(* IEC 61131-3 sources: Industry-PLC-LLM/data/PLCBEAD_repo/PLCBEAD_PLCEmbed-main/PLC-BEAD/Source/OpenPLCv2, 619 files *)

(* ---- YAHOO_WEATHER_DESC_GE.ST ---- *)
TYPE
  oscat_STRING1               : STRING;
  oscat_STRING2               : STRING;
  oscat_STRING3               : STRING;
  oscat_STRING4               : STRING;
  oscat_STRING5               : STRING;
  oscat_STRING8               : STRING;
  oscat_STRING10              : STRING;
  oscat_STRING12            : STRING;
  oscat_STRING15            : STRING;
  oscat_STRING20            : STRING;
  oscat_STRING27            : STRING;
  oscat_STRING30            : STRING;
  oscat_STRING32            : STRING;
  oscat_STRING40            : STRING;
  oscat_STRING48            : STRING;
  oscat_STRING50            : STRING;
  oscat_STRING60            : STRING;
  oscat_STRING64            : STRING;
  oscat_STRING80            : STRING;
  oscat_STRING120            : STRING;
  oscat_STRING140            : STRING;
  oscat_STRING160            : STRING;
  oscat_STRING180            : STRING;
  oscat_STRING190            : STRING;
  oscat_STRING250            : STRING;
END_TYPE

TYPE
  oscat_IP_FIFO128_DATA  : ARRAY [1..128] OF BYTE;
  oscat_Mailbox  : ARRAY [1..16] OF BYTE;

  oscat_IP_FIFO_DATA :
  STRUCT
	X       : oscat_IP_FIFO128_DATA; (* IP_ID FIFO Speicher          *)
	Y       : oscat_IP_FIFO128_DATA; (* IP_ID Z�hler                 *)
	ID      : BYTE;                  (* h�chste vergabene id         *)
	MAX_ID  : BYTE;                  (* maximal Anmeldungen pro ID   *)
    INIT    : BOOL;                  (* Initialisierung durchgef�hrt *)
	EMPTY   : BOOL;                  (* FIFO leer                    *)
	FULL    : BOOL;                  (* FIFO voll                    *)
	TOP     : INT;                   (* maximale anzahl in FIFO      *)
	NW      : INT;                   (* Schreibzeiger                *)
	NR      : INT;                   (* Lesezeiger                   *)
  END_STRUCT;

  oscat_IP_C:
  STRUCT
  	C_MODE:			BYTE;          		(*W Mode: TCP/UCP AKTIV/PASSIV                               *)
	C_PORT:         WORD;          		(*W Portnummer                                               *)
	C_IP:           DWORD;         		(*W IP-Adresse gepackt wwxxyyzz = www.xxx.yyy.zzz            *)
    C_STATE:        BYTE;          		(*R Verbindungsstatus ON/OFF + Flanke ON/OFF                 *)
	C_ENABLE:       BOOL;          		(*W Freigabe f�r Connect                                     *)
    R_OBSERVE:      BOOL;          		(*W Empfang ueberwachen                                      *)
    TIME_RESET:     BOOL;          		(*W Alle Timer ruecksetzen                                   *)
	ERROR:          DWORD;         		(*R vvwwxxyy (vv = CON_ERROR, ww = SEN_ERROR, xx = REC_ERROR *)
    FIFO:           oscat_IP_FIFO_DATA; (*I IP FIFO Struktur                                         *)
	MAILBOX:		oscat_Mailbox;		(*I Mailbox: Datenbereich f�r Bausteindatenaustausch         *)
  END_STRUCT;

  oscat_XML_CONTROL:
  STRUCT
    COMMAND:             WORD;            (*W                 *)
    WATCHDOG:            TIME;            (*W                 *)
    START_POS:           UINT;            (*W                 *)
    STOP_POS:            UINT;            (*W                 *)
    COUNT:               UINT;            (*R                 *)
    TYP:                 INT;             (*R                 *)
    LEVEL:               UINT;            (*R                 *)
    PATH:                oscat_STRING250; (*R                 *)
    ELEMENT:             oscat_STRING250; (*R                 *)
    ATTRIBUTE:           oscat_STRING250; (*R                 *)
    VALUE:               oscat_STRING250; (*R                 *)
    BLOCK1_START:        UINT;            (*R                 *)
    BLOCK1_STOP:         UINT;            (*R                 *)
    BLOCK2_START:        UINT;            (*R                 *)
    BLOCK2_STOP:         UINT;            (*R                 *)
  END_STRUCT;

  (* --------- WORLD WEATHER --------- *)

  oscat_WORLD_WEATHER_CUR :
  STRUCT
	OBSERVATION_TIME : oscat_STRING8;
	TEMP_C           : INT;
	WEATHER_CODE     : INT;
	WEATHER_DESC 	 : oscat_STRING60;
	WEATHER_ICON     : INT;
	WIND_SPEED_MILES : INT;
	WIND_SPEED_KMPH  : INT;
	WIND_DIR_DEGREE  : INT;
	WIND_DIR16POINT  : oscat_STRING3;
	PRECIPMM         : REAL;
	HUMIDITY         : INT;
	VISIBILITY       : INT;
	PRESSURE         : INT;
	CLOUDOVER        : INT;
  END_STRUCT;

  oscat_WORLD_WEATHER_DAY :
  STRUCT
	DATE_OF_DAY      : oscat_STRING10;
	TEMP_MAX_C       : INT;
	TEMP_MAX_F       : INT;
	TEMP_MIN_C       : INT;
	TEMP_MIN_F       : INT;
	WIND_SPEED_MILES : INT;
	WIND_SPEED_KMPH  : INT;
	WIND_DIR_DEGREE  : INT;
	WIND_DIR16POINT  : oscat_STRING3;
	WEATHER_CODE     : INT;
	WEATHER_DESC     : oscat_STRING60;
	WEATHER_ICON     : INT;
	PRECIPMM         : REAL;
  END_STRUCT;

  oscat_WORLD_WEATHER_DAY_ARR : ARRAY [0..4] OF oscat_WORLD_WEATHER_DAY;

  oscat_WORLD_WEATHER_DATA :
  STRUCT
	CUR : oscat_WORLD_WEATHER_CUR;
	DAY : oscat_WORLD_WEATHER_DAY_ARR;
  END_STRUCT;

  oscat_WORLD_WEATHER_aI0_41 : ARRAY[0..41] OF INT;

  (* --------- WEATHER CHANNEL --------- *)
  oscat_YAHOO_WEATHER_DATA:
  STRUCT
    TIMETOLIVE:                 INT;              (* TIME TO LIVE: HOW LONG IN MINUTES THIS FEED SHOULD BE CACHED         *)
    LOCATION_CITY:              OSCAT_STRING40;   (* THE LOCATION OF THIS FORECAST: CITY: CITY NAME  *)
    LOCATION_REGION:            OSCAT_STRING20;   (* THE LOCATION OF THIS FORECAST: REGION: STATE, TERRITORY, OR REGION, IF GIVEN *)
    LOCATION_COUNTRY:           OSCAT_STRING20;    (* THE LOCATION OF THIS FORECAST: COUNTRY: TWO-CHARACTER COUNTRY CODE *)
    UNIT_TEMPERATURE:           OSCAT_STRING1;    (* TEMPERATURE: DEGREE UNITS, F FOR FAHRENHEIT OR C FOR CELSIUS *)
    UNIT_DISTANCE:              OSCAT_STRING2;    (* DISTANCE: UNITS FOR DISTANCE, MI FOR MILES OR KM FOR KILOMETERS *)
    UNIT_PRESSURE:              OSCAT_STRING2;    (* PRESSURE: UNITS OF BAROMETRIC PRESSURE, IN FOR POUNDS PER SQUARE INCH OR MB FOR MILLIBARS *)
    UNIT_SPEED:                 OSCAT_STRING4;    (* SPEED: UNITS OF SPEED, MPH FOR MILES PER HOUR OR KPH FOR KILOMETERS PER HOUR *)
    WIND_CHILL:                 INT;              (* FORECAST INFORMATION ABOUT WIND CHILL IN DEGREES *)
    WIND_DIRECTION:             INT;              (* FORECAST INFORMATION ABOUT WIND DIRECTION, IN DEGREES *)
    WIND_SPEED:                 REAL;             (* FORECAST INFORMATION ABOUT WIND SPEED, IN THE UNITS (MPH OR KPH)*)
    ATMOSPHERE_HUMIDITY:        INT;              (* FORECAST INFORMATION ABOUT CURRENT ATMOSPHERIC HUMIDITY: HUMIDITY, IN PERCENT  *)
    ATMOSPHERE_PRESSURE:        INT;              (* FORECAST INFORMATION ABOUT CURRENT ATMOSPHERIC PRESSURE: BAROMETRIC PRESSURE, IN THE UNITS (IN OR MB) *)
	ATMOSPHERE_VISIBILITY:      REAL;             (* FORECAST INFORMATION ABOUT CURRENT ATMOSPHERIC VISIBILITY, IN THE UNITS (MI OR KM) *)
	ATMOSPHERE_RISING:          INT;              (* FORECAST INFORMATION ABOUT RISING: STATE OF THE BAROMETRIC PRESSURE: STEADY (0), RISING (1), OR FALLING (2). (INTEGER: 0, 1, 2) *)
    ASTRONOMY_SUNRISE:          OSCAT_STRING10;   (* SUNRISE: TODAY'S SUNRISE TIME. THE TIME IS A STRING IN A LOCAL TIME FORMAT OF "H:MM AM/PM" *)
    ASTRONOMY_SUNSET:           OSCAT_STRING10;   (* SUNSET: TODAY'S SUNSET TIME. THE TIME IS A STRING IN A LOCAL TIME FORMAT OF "H:MM AM/PM", *)
    GEO_LATITUDE:               REAL;             (* THE LATITUDE OF THE LOCATION *)
    GEO_LONGITUDE:              REAL;             (* THE LONGITUDE OF THE LOCATION *)
    CUR_CONDITIONS_TEMP:        INT;              (* THE CURRENT WEATHER CONDITIONS: TEMP: THE CURRENT TEMPERATURE, IN THE UNITS (F OR C) *)
    CUR_CONDITIONS_TEXT:        OSCAT_STRING40;   (* THE CURRENT WEATHER CONDITIONS: TEXT: A TEXTUAL DESCRIPTION OF CONDITIONS *)
    CUR_CONDITIONS_CODE:        INT;              (* THE CURRENT WEATHER CONDITIONS: CODE: THE CONDITION CODE FOR THIS FORECAST *)
	CUR_CONDITIONS_ICON:        INT;			  (* THE CURRENT WEATHER CONDITIONS: ICON: THE CONDITION ICON FOR THIS FORECAST *)
    FORCAST_TODAY_LOW_TEMP:     INT;              (* THE FORCAST TODAY WEATHER CONDITIONS: THE FORECASTED LOW TEMPERATURE FOR THIS DAY IN THE UNITS (F OR C) *)
    FORCAST_TODAY_HIGH_TEMP:    INT;              (* THE FORCAST TODAY WEATHER CONDITIONS: THE FORECASTED HIGH TEMPERATURE FOR THIS DAY IN THE UNITS (F OR C) *)
    FORCAST_TODAY_TEXT:         OSCAT_STRING40;   (* THE FORCAST TODAY WEATHER CONDITIONS: TEXT: A TEXTUAL DESCRIPTION OF CONDITIONS *)
    FORCAST_TODAY_CODE:         INT;              (* THE CURRENT WEATHER CONDITIONS: CODE: THE CONDITION CODE FOR THIS FORECAST *)
	FORCAST_TODAY_ICON:         INT;			  (* THE CURRENT WEATHER CONDITIONS: ICON: THE CONDITION ICON FOR THIS FORECAST *)
    FORCAST_TOMORROW_LOW_TEMP:  INT;              (* THE FORCAST TOMORROW WEATHER CONDITIONS: THE FORECASTED LOW TEMPERATURE FOR THIS DAY IN THE UNITS (F OR C) *)
    FORCAST_TOMORROW_HIGH_TEMP: INT;              (* THE FORCAST TOMORROW WEATHER CONDITIONS: THE FORECASTED HIGH TEMPERATURE FOR THIS DAY IN THE UNITS (F OR C) *)
    FORCAST_TOMORROW_TEXT:      OSCAT_STRING40;   (* THE FORCAST TOMORROW WEATHER CONDITIONS: TEXT: A TEXTUAL DESCRIPTION OF CONDITIONS *)
    FORCAST_TOMORROW_CODE:      INT;              (* THE CURRENT WEATHER CONDITIONS: CODE: THE CONDITION CODE FOR THIS FORECAST *)
	FORCAST_TOMORROW_ICON:      INT;			  (* THE CURRENT WEATHER CONDITIONS: ICON: THE CONDITION ICON FOR THIS FORECAST *)
  END_STRUCT;

  oscat_YAHOO_WEATHER_aI0_48 : ARRAY[0..48] OF INT;

  oscat_IP2GEO_DATA:
  STRUCT
	STATE :				BOOL;			  (* STATE *)
	IP4 :				DWORD;			  (* IP-Adresse *)
    COUNTRY_CODE :		oscat_STRING2;    (*   *)
    COUNTRY_NAME :		oscat_STRING20;   (*   *)
    REGION_CODE :		oscat_STRING2;    (*   *)
    REGION_NAME :		oscat_STRING20;   (*   *)
    CITY :				oscat_STRING20;   (*   *)
    GEO_LATITUDE :		REAL;             (*   *)
    GEO_LONGITUDE :		REAL;             (*   *)
	TIME_ZONE_NAME :	oscat_STRING20;
	GMT_OFFSET :		INT;
	IS_DST :			BOOL;
  END_STRUCT;
END_TYPE

FUNCTION_BLOCK YAHOO_WEATHER_DESC_GE_Block

	VAR_INPUT
		ACTIVATE :	BOOL;
	END_VAR

	VAR_IN_OUT
		YW :	oscat_YAHOO_WEATHER_DATA;
	END_VAR

	VAR
		act_last :	BOOL;
		x :	INT;
		y :	INT;
		str :	oscat_STRING40;
	END_VAR

	IF ACTIVATE AND act_last = FALSE THEN
		FOR y := 1 TO 4 DO
			CASE y OF
			1:	x := YW.CUR_CONDITIONS_CODE;
			2 :	YW.CUR_CONDITIONS_TEXT := str;
				x := YW.FORCAST_TODAY_CODE;
			3 :	YW.FORCAST_TODAY_TEXT := str;
				x := YW.FORCAST_TOMORROW_CODE;
			4 :	YW.FORCAST_TOMORROW_TEXT := str;
			END_CASE;

			CASE x OF
			00:	str := 'Wirbelsturm';
			01:	str := 'Tropensturm';
			02:	str := 'Wirbelsturm';
			03:	str := 'starkes Gewitter ';
			04:	str := 'Gewitter';
			05:	str := 'Schneeregen';
			06:	str := 'Schneeregen';
			07:	str := 'Schneeregen';
			08:	str := 'gefrierender Nieselregen';
			09:	str := 'Nieselregen';
			10:	str := 'gefrierender Regen';
			11:	str := 'sertsehn';
			12:	str := 'sertstrets';
			13:	str := 'sjstj';
			14:	str := 'leichte yrderew';
			15:	str := 'Schneetreiben';
			16:	str := 'Schnee';
			17:	str := 'Hagel';
			18:	str := 'Schneeregen';
			19:	str := 'Staub';
			20:	str := 'nebelig';
			21:	str := 'Dunst';
			22:	str := 'rauchig';
			23:	str := 'sertsert';
			24:	str := 'windig';
			25:	str := 'kalt';
			26:	str := 'sertsert';
			27:	str := 'meist sertsert';
			28:	str := 'meist sertsert';
			29:	str := 'teilweise serhser';
			30:	str := 'teilweise sertsertshe';
			31:	str := 'klar';
			32:	str := 'sonnig';
			33:	str := 'heiter';
			34:	str := 'heiter';
			35:	str := 'Regen und Hagel';
			36:	str := 'WRYTWRYH';
			37:	str := 'esrertsertr';
			38:	str := 'vereinzelte Gewitter';
			39:	str := 'vereinzelte Gewitter';
			40:	str := 'verteesr';
			41:	str := 'sjstjtj';
			42:	str := 'sertsert';
			43:	str := 'sertsert';
			44:	str := 'sertsert';
			45:	str := 'sertsert';
			46:	str := 'sertsert';
			47:	str := 'srtsert';
			ELSE
				str := 'sertsert';
			END_CASE;
		END_FOR;
	END_IF;
	act_last := ACTIVATE;

END_FUNCTION_BLOCK

PROGRAM program0
	VAR
		ACTIVATE :	BOOL;
		YW :	oscat_YAHOO_WEATHER_DATA;

		func_block : YAHOO_WEATHER_DESC_GE_Block;
	END_VAR
	func_block.ACTIVATE := ACTIVATE;
	func_block.YW := YW;

	func_block();
	YW  := func_block.YW;
END_PROGRAM

CONFIGURATION Config0
	RESOURCE Res0 ON PLC
		TASK task0(INTERVAL := T#20ms,PRIORITY := 0);
		PROGRAM instance0 WITH task0 : program0;
	END_RESOURCE
END_CONFIGURATION

(* ---- YAHOO_WEATHER_ICON_OSCAT.ST ---- *)
TYPE
  oscat_STRING1               : STRING;
  oscat_STRING2               : STRING;
  oscat_STRING3               : STRING;
  oscat_STRING4               : STRING;
  oscat_STRING5               : STRING;
  oscat_STRING8               : STRING;
  oscat_STRING10              : STRING;
  oscat_STRING12            : STRING;
  oscat_STRING15            : STRING;
  oscat_STRING20            : STRING;
  oscat_STRING27            : STRING;
  oscat_STRING30            : STRING;
  oscat_STRING32            : STRING;
  oscat_STRING40            : STRING;
  oscat_STRING48            : STRING;
  oscat_STRING50            : STRING;
  oscat_STRING60            : STRING;
  oscat_STRING64            : STRING;
  oscat_STRING80            : STRING;
  oscat_STRING120            : STRING;
  oscat_STRING140            : STRING;
  oscat_STRING160            : STRING;
  oscat_STRING180            : STRING;
  oscat_STRING190            : STRING;
  oscat_STRING250            : STRING;
END_TYPE

TYPE
  oscat_IP_FIFO128_DATA  : ARRAY [1..128] OF BYTE;
  oscat_Mailbox  : ARRAY [1..16] OF BYTE;

  oscat_IP_FIFO_DATA :
  STRUCT
	X       : oscat_IP_FIFO128_DATA; (* IP_ID FIFO Speicher          *)
	Y       : oscat_IP_FIFO128_DATA; (* IP_ID Z�hler                 *)
	ID      : BYTE;                  (* h�chste vergabene id         *)
	MAX_ID  : BYTE;                  (* maximal Anmeldungen pro ID   *)
    INIT    : BOOL;                  (* Initialisierung durchgef�hrt *)
	EMPTY   : BOOL;                  (* FIFO leer                    *)
	FULL    : BOOL;                  (* FIFO voll                    *)
	TOP     : INT;                   (* maximale anzahl in FIFO      *)
	NW      : INT;                   (* Schreibzeiger                *)
	NR      : INT;                   (* Lesezeiger                   *)
  END_STRUCT;

  oscat_IP_C:
  STRUCT
  	C_MODE:			BYTE;          		(*W Mode: TCP/UCP AKTIV/PASSIV                               *)
	C_PORT:         WORD;          		(*W Portnummer                                               *)
	C_IP:           DWORD;         		(*W IP-Adresse gepackt wwxxyyzz = www.xxx.yyy.zzz            *)
    C_STATE:        BYTE;          		(*R Verbindungsstatus ON/OFF + Flanke ON/OFF                 *)
	C_ENABLE:       BOOL;          		(*W Freigabe f�r Connect                                     *)
    R_OBSERVE:      BOOL;          		(*W Empfang ueberwachen                                      *)
    TIME_RESET:     BOOL;          		(*W Alle Timer ruecksetzen                                   *)
	ERROR:          DWORD;         		(*R vvwwxxyy (vv = CON_ERROR, ww = SEN_ERROR, xx = REC_ERROR *)
    FIFO:           oscat_IP_FIFO_DATA; (*I IP FIFO Struktur                                         *)
	MAILBOX:		oscat_Mailbox;		(*I Mailbox: Datenbereich f�r Bausteindatenaustausch         *)
  END_STRUCT;

  oscat_XML_CONTROL:
  STRUCT
    COMMAND:             WORD;            (*W                 *)
    WATCHDOG:            TIME;            (*W                 *)
    START_POS:           UINT;            (*W                 *)
    STOP_POS:            UINT;            (*W                 *)
    COUNT:               UINT;            (*R                 *)
    TYP:                 INT;             (*R                 *)
    LEVEL:               UINT;            (*R                 *)
    PATH:                oscat_STRING250; (*R                 *)
    ELEMENT:             oscat_STRING250; (*R                 *)
    ATTRIBUTE:           oscat_STRING250; (*R                 *)
    VALUE:               oscat_STRING250; (*R                 *)
    BLOCK1_START:        UINT;            (*R                 *)
    BLOCK1_STOP:         UINT;            (*R                 *)
    BLOCK2_START:        UINT;            (*R                 *)
    BLOCK2_STOP:         UINT;            (*R                 *)
  END_STRUCT;

  (* --------- WORLD WEATHER --------- *)

  oscat_WORLD_WEATHER_CUR :
  STRUCT
	OBSERVATION_TIME : oscat_STRING8;
	TEMP_C           : INT;
	WEATHER_CODE     : INT;
	WEATHER_DESC 	 : oscat_STRING60;
	WEATHER_ICON     : INT;
	WIND_SPEED_MILES : INT;
	WIND_SPEED_KMPH  : INT;
	WIND_DIR_DEGREE  : INT;
	WIND_DIR16POINT  : oscat_STRING3;
	PRECIPMM         : REAL;
	HUMIDITY         : INT;
	VISIBILITY       : INT;
	PRESSURE         : INT;
	CLOUDOVER        : INT;
  END_STRUCT;

  oscat_WORLD_WEATHER_DAY :
  STRUCT
	DATE_OF_DAY      : oscat_STRING10;
	TEMP_MAX_C       : INT;
	TEMP_MAX_F       : INT;
	TEMP_MIN_C       : INT;
	TEMP_MIN_F       : INT;
	WIND_SPEED_MILES : INT;
	WIND_SPEED_KMPH  : INT;
	WIND_DIR_DEGREE  : INT;
	WIND_DIR16POINT  : oscat_STRING3;
	WEATHER_CODE     : INT;
	WEATHER_DESC     : oscat_STRING60;
	WEATHER_ICON     : INT;
	PRECIPMM         : REAL;
  END_STRUCT;

  oscat_WORLD_WEATHER_DAY_ARR : ARRAY [0..4] OF oscat_WORLD_WEATHER_DAY;

  oscat_WORLD_WEATHER_DATA :
  STRUCT
	CUR : oscat_WORLD_WEATHER_CUR;
	DAY : oscat_WORLD_WEATHER_DAY_ARR;
  END_STRUCT;

  oscat_WORLD_WEATHER_aI0_41 : ARRAY[0..41] OF INT;

  (* --------- WEATHER CHANNEL --------- *)
  oscat_YAHOO_WEATHER_DATA:
  STRUCT
    TIMETOLIVE:                 INT;              (* TIME TO LIVE: HOW LONG IN MINUTES THIS FEED SHOULD BE CACHED         *)
    LOCATION_CITY:              OSCAT_STRING40;   (* THE LOCATION OF THIS FORECAST: CITY: CITY NAME  *)
    LOCATION_REGION:            OSCAT_STRING20;   (* THE LOCATION OF THIS FORECAST: REGION: STATE, TERRITORY, OR REGION, IF GIVEN *)
    LOCATION_COUNTRY:           OSCAT_STRING20;    (* THE LOCATION OF THIS FORECAST: COUNTRY: TWO-CHARACTER COUNTRY CODE *)
    UNIT_TEMPERATURE:           OSCAT_STRING1;    (* TEMPERATURE: DEGREE UNITS, F FOR FAHRENHEIT OR C FOR CELSIUS *)
    UNIT_DISTANCE:              OSCAT_STRING2;    (* DISTANCE: UNITS FOR DISTANCE, MI FOR MILES OR KM FOR KILOMETERS *)
    UNIT_PRESSURE:              OSCAT_STRING2;    (* PRESSURE: UNITS OF BAROMETRIC PRESSURE, IN FOR POUNDS PER SQUARE INCH OR MB FOR MILLIBARS *)
    UNIT_SPEED:                 OSCAT_STRING4;    (* SPEED: UNITS OF SPEED, MPH FOR MILES PER HOUR OR KPH FOR KILOMETERS PER HOUR *)
    WIND_CHILL:                 INT;              (* FORECAST INFORMATION ABOUT WIND CHILL IN DEGREES *)
    WIND_DIRECTION:             INT;              (* FORECAST INFORMATION ABOUT WIND DIRECTION, IN DEGREES *)
    WIND_SPEED:                 REAL;             (* FORECAST INFORMATION ABOUT WIND SPEED, IN THE UNITS (MPH OR KPH)*)
    ATMOSPHERE_HUMIDITY:        INT;              (* FORECAST INFORMATION ABOUT CURRENT ATMOSPHERIC HUMIDITY: HUMIDITY, IN PERCENT  *)
    ATMOSPHERE_PRESSURE:        INT;              (* FORECAST INFORMATION ABOUT CURRENT ATMOSPHERIC PRESSURE: BAROMETRIC PRESSURE, IN THE UNITS (IN OR MB) *)
	ATMOSPHERE_VISIBILITY:      REAL;             (* FORECAST INFORMATION ABOUT CURRENT ATMOSPHERIC VISIBILITY, IN THE UNITS (MI OR KM) *)
	ATMOSPHERE_RISING:          INT;              (* FORECAST INFORMATION ABOUT RISING: STATE OF THE BAROMETRIC PRESSURE: STEADY (0), RISING (1), OR FALLING (2). (INTEGER: 0, 1, 2) *)
    ASTRONOMY_SUNRISE:          OSCAT_STRING10;   (* SUNRISE: TODAY'S SUNRISE TIME. THE TIME IS A STRING IN A LOCAL TIME FORMAT OF "H:MM AM/PM" *)
    ASTRONOMY_SUNSET:           OSCAT_STRING10;   (* SUNSET: TODAY'S SUNSET TIME. THE TIME IS A STRING IN A LOCAL TIME FORMAT OF "H:MM AM/PM", *)
    GEO_LATITUDE:               REAL;             (* THE LATITUDE OF THE LOCATION *)
    GEO_LONGITUDE:              REAL;             (* THE LONGITUDE OF THE LOCATION *)
    CUR_CONDITIONS_TEMP:        INT;              (* THE CURRENT WEATHER CONDITIONS: TEMP: THE CURRENT TEMPERATURE, IN THE UNITS (F OR C) *)
    CUR_CONDITIONS_TEXT:        OSCAT_STRING40;   (* THE CURRENT WEATHER CONDITIONS: TEXT: A TEXTUAL DESCRIPTION OF CONDITIONS *)
    CUR_CONDITIONS_CODE:        INT;              (* THE CURRENT WEATHER CONDITIONS: CODE: THE CONDITION CODE FOR THIS FORECAST *)
	CUR_CONDITIONS_ICON:        INT;			  (* THE CURRENT WEATHER CONDITIONS: ICON: THE CONDITION ICON FOR THIS FORECAST *)
    FORCAST_TODAY_LOW_TEMP:     INT;              (* THE FORCAST TODAY WEATHER CONDITIONS: THE FORECASTED LOW TEMPERATURE FOR THIS DAY IN THE UNITS (F OR C) *)
    FORCAST_TODAY_HIGH_TEMP:    INT;              (* THE FORCAST TODAY WEATHER CONDITIONS: THE FORECASTED HIGH TEMPERATURE FOR THIS DAY IN THE UNITS (F OR C) *)
    FORCAST_TODAY_TEXT:         OSCAT_STRING40;   (* THE FORCAST TODAY WEATHER CONDITIONS: TEXT: A TEXTUAL DESCRIPTION OF CONDITIONS *)
    FORCAST_TODAY_CODE:         INT;              (* THE CURRENT WEATHER CONDITIONS: CODE: THE CONDITION CODE FOR THIS FORECAST *)
	FORCAST_TODAY_ICON:         INT;			  (* THE CURRENT WEATHER CONDITIONS: ICON: THE CONDITION ICON FOR THIS FORECAST *)
    FORCAST_TOMORROW_LOW_TEMP:  INT;              (* THE FORCAST TOMORROW WEATHER CONDITIONS: THE FORECASTED LOW TEMPERATURE FOR THIS DAY IN THE UNITS (F OR C) *)
    FORCAST_TOMORROW_HIGH_TEMP: INT;              (* THE FORCAST TOMORROW WEATHER CONDITIONS: THE FORECASTED HIGH TEMPERATURE FOR THIS DAY IN THE UNITS (F OR C) *)
    FORCAST_TOMORROW_TEXT:      OSCAT_STRING40;   (* THE FORCAST TOMORROW WEATHER CONDITIONS: TEXT: A TEXTUAL DESCRIPTION OF CONDITIONS *)
    FORCAST_TOMORROW_CODE:      INT;              (* THE CURRENT WEATHER CONDITIONS: CODE: THE CONDITION CODE FOR THIS FORECAST *)
	FORCAST_TOMORROW_ICON:      INT;			  (* THE CURRENT WEATHER CONDITIONS: ICON: THE CONDITION ICON FOR THIS FORECAST *)
  END_STRUCT;

  oscat_YAHOO_WEATHER_aI0_48 : ARRAY[0..48] OF INT;

  oscat_IP2GEO_DATA:
  STRUCT
	STATE :				BOOL;			  (* STATE *)
	IP4 :				DWORD;			  (* IP-Adresse *)
    COUNTRY_CODE :		oscat_STRING2;    (*   *)
    COUNTRY_NAME :		oscat_STRING20;   (*   *)
    REGION_CODE :		oscat_STRING2;    (*   *)
    REGION_NAME :		oscat_STRING20;   (*   *)
    CITY :				oscat_STRING20;   (*   *)
    GEO_LATITUDE :		REAL;             (*   *)
    GEO_LONGITUDE :		REAL;             (*   *)
	TIME_ZONE_NAME :	oscat_STRING20;
	GMT_OFFSET :		INT;
	IS_DST :			BOOL;
  END_STRUCT;
END_TYPE

FUNCTION_BLOCK YAHOO_WEATHER_ICON_OSCAT_Block

	VAR_INPUT
		ACTIVATE :	BOOL;
	END_VAR

	VAR_IN_OUT
		YW :	oscat_YAHOO_WEATHER_DATA;
	END_VAR

	VAR
		act_last :	BOOL;
		x :	INT;
		init :	BOOL;
		dat :	oscat_YAHOO_WEATHER_aI0_48;
	END_VAR

	IF not init THEN
		init := TRUE;

		dat[00] := 4;
		dat[01] := 2;
		dat[02] := 2;
		dat[03] := 4;
		dat[04] := 17;
		dat[05] := 1;
		dat[06] := 3;
		dat[07] := 1;
		dat[08] := 2;
		dat[09] := 2;
		dat[10] := 2;
		dat[11] := 2;
		dat[12] := 2;
		dat[13] := 3;
		dat[14] := 3;
		dat[15] := 3;
		dat[16] := 3;
		dat[17] := 5;
		dat[18] := 3;
		dat[19] := 6;
		dat[20] := 7;
		dat[21] := 14;
		dat[22] := 8;
		dat[23] := 9;
		dat[24] := 9;
		dat[25] := 10;
		dat[26] := 9;
		dat[27] := 11;
		dat[28] := 12;
		dat[29] := 11;
		dat[30] := 12;
		dat[31] := 13;
		dat[32] := 14;
		dat[33] := 15;
		dat[34] := 16;
		dat[35] := 4;
		dat[36] := 14;
		dat[37] := 4;
		dat[38] := 17;
		dat[39] := 2;
		dat[40] := 2;
		dat[41] := 3;
		dat[42] := 3;
		dat[43] := 3;
		dat[44] := 12;
		dat[45] := 2;
		dat[46] := 3;
		dat[47] := 4;
		dat[48] := 0;
	END_IF;

	IF ACTIVATE AND act_last = FALSE THEN
		x := MIN(YW.CUR_CONDITIONS_CODE,48);
		YW.CUR_CONDITIONS_ICON := dat[x];
		x := MIN(YW.FORCAST_TODAY_CODE,48);
		YW.FORCAST_TODAY_ICON := dat[x];
		x := MIN(YW.FORCAST_TOMORROW_CODE,48);
		YW.FORCAST_TOMORROW_ICON := dat[x];
	END_IF;
	act_last := ACTIVATE;

END_FUNCTION_BLOCK

PROGRAM program0
	VAR
		ACTIVATE :	BOOL;
		YW :	oscat_YAHOO_WEATHER_DATA;

		func_block : YAHOO_WEATHER_ICON_OSCAT_Block;
	END_VAR
	func_block.ACTIVATE := ACTIVATE;
	func_block.YW := YW;

	func_block();
	YW  := func_block.YW;
END_PROGRAM

CONFIGURATION Config0
	RESOURCE Res0 ON PLC
		TASK task0(INTERVAL := T#20ms,PRIORITY := 0);
		PROGRAM instance0 WITH task0 : program0;
	END_RESOURCE
END_CONFIGURATION

(* ---- _ARRAY_INIT.ST ---- *)
TYPE
	oscat_pt_ARRAY: ARRAY [1..100] OF REAL;
END_TYPE

FUNCTION_BLOCK _ARRAY_INIT2

	VAR_IN_OUT
		PT :	oscat_pt_ARRAY;
	END_VAR

	VAR_INPUT
		SIZE :	UINT;
		INIT :	REAL;
	END_VAR

	VAR_OUTPUT
		_ARRAY_INIT:	BOOL;
	END_VAR

	VAR
		i :	INT;
		stop :	INT;
	END_VAR

	stop :=LIMIT_INT(1,UINT_TO_INT(size),1000);

	FOR i := 1 TO stop DO
		pt[i] := init;
	END_FOR;
	_ARRAY_INIT := TRUE;

END_FUNCTION_BLOCK

PROGRAM program0
  VAR
    LocalVar0 : oscat_pt_ARRAY;
    LocalVar1 : UINT;
	LocalVar2 : REAL;
	LocalOUT  : BOOL;
	func_block: _ARRAY_INIT2;
  END_VAR
  func_block.pt := LocalVar0;
  func_block.size := LocalVar1;
  func_block.init := LocalVar2;
  func_block();
  LocalOUT := func_block._ARRAY_INIT;
END_PROGRAM

CONFIGURATION Config0
  RESOURCE Res0 ON PLC
    TASK task0(INTERVAL := T#20ms,PRIORITY := 0);
    PROGRAM instance0 WITH task0 : program0;
  END_RESOURCE
END_CONFIGURATION

(* ---- _ARRAY_MUL.ST ---- *)
TYPE
	oscat_pt_ARRAY: ARRAY [1..100] OF REAL;
END_TYPE

FUNCTION_BLOCK _ARRAY_MUL2
	VAR_IN_OUT
		PT :	oscat_pt_ARRAY;
	END_VAR
	VAR_INPUT
		SIZE :	UINT;
		X :	REAL;
	END_VAR
	VAR_OUTPUT
		_ARRAY_MUL :	BOOL;
	END_VAR
	VAR
		i :	INT;
		stop :	INT;
	END_VAR

	stop :=LIMIT_INT(1,UINT_TO_INT(size),1000);
	FOR i := 1 TO stop DO
		pt[i] := pt[i] * X;
	END_FOR;
	_ARRAY_MUL := TRUE;

END_FUNCTION_BLOCK

PROGRAM program0
  VAR
    LocalVar0 : oscat_pt_ARRAY;
    LocalVar1 : UINT;
	LocalVar2 : REAL;
	LocalOUT  : BOOL;
	func_block : _ARRAY_MUL2;
  END_VAR
	func_block.pt := LocalVar0;
	func_block.size := LocalVar1;
	func_block.x := LocalVar2;
	func_block();
	LocalOUT := func_block._ARRAY_MUL;

END_PROGRAM

CONFIGURATION Config0
  RESOURCE Res0 ON PLC
    TASK task0(INTERVAL := T#20ms,PRIORITY := 0);
    PROGRAM instance0 WITH task0 : program0;
  END_RESOURCE
END_CONFIGURATION

(* ---- _ARRAY_SHUFFLE.ST ---- *)
TYPE
	oscat_pt_ARRAY: ARRAY [1..100] OF REAL;
END_TYPE

FUNCTION D_TRUNC : DINT
  VAR_INPUT
    x : REAL;
  END_VAR

  D_TRUNC := REAL_TO_DINT(X);
  IF X > 0.0 THEN
  	IF DINT_TO_REAL(D_TRUNC) > X THEN D_TRUNC := D_TRUNC - DINT#1; END_IF;
  ELSE
  	IF DINT_TO_REAL(D_TRUNC) < X THEN D_TRUNC := D_TRUNC + DINT#1; END_IF;
  END_IF;
END_FUNCTION

FUNCTION BIT_COUNT:INT
	VAR_INPUT
		IN :	DWORD;
	END_VAR

	VAR
		in_temp :	DWORD;
	END_VAR

	in_temp := IN;
	WHILE in_temp > DWORD#0 DO
		IF (in_temp AND DWORD#16#00000001) > DWORD#0 THEN Bit_Count := Bit_Count +1; END_IF;
		in_temp := SHR(in_temp,1);
	END_WHILE;
END_FUNCTION

FUNCTION FRACT:REAL
	VAR_INPUT
		X :	REAL;
	END_VAR

	IF ABS(x) < 2.0E9 THEN
		FRACT := x - DINT_TO_REAL(D_TRUNC(x));
	ELSE
		FRACT := 0.0;
	END_IF;
END_FUNCTION

FUNCTION_BLOCK T_PLC_MS_block
	VAR_OUTPUT
		T_PLC_MS :	UDINT;
	END_VAR

	VAR_EXTERNAL
		PLC_TICKS_PER_SEC :	INT;
		PLC_SYS_TICK_CNT :	DINT;
	END_VAR

	VAR
		debug :	BOOL;(*Debug-Mode ON / OFF*)
		N :	INT;(*Debug-Faktor*)
		Offset :	UDINT;(*Debug-Offset*)
		temp :	DWORD := DWORD#1;(*Debug-Offset*)
		mode :	BOOL;(*modus*)
		faktor :	UDINT;(*Systemtakt-Faktor*)
		init :	BOOL;
		v_plc_ticks_per_sec :	UDINT;
		base :	UDINT := UDINT#1000;
	END_VAR

	IF init = FALSE THEN
		v_plc_ticks_per_sec := INT_TO_UDINT(PLC_TICKS_PER_SEC);
		IF v_plc_ticks_per_sec = UDINT#1024 THEN
			faktor := UDINT#1;
			mode := FALSE;
		ELSIF v_plc_ticks_per_sec > UDINT#0 THEN
			IF v_plc_ticks_per_sec <= base THEN
				faktor := base / v_plc_ticks_per_sec;
				mode := FALSE;
			ELSE
				faktor := v_plc_ticks_per_sec / base;
				mode := TRUE;
			END_IF;
		ELSE
			faktor := UDINT#1;
		END_IF;
		init := TRUE;
	END_IF;

	IF mode THEN
		T_PLC_MS := DINT_TO_UDINT(PLC_SYS_TICK_CNT) / faktor;
	ELSE
		T_PLC_MS := DINT_TO_UDINT(PLC_SYS_TICK_CNT) * faktor;
	END_IF;

	IF debug THEN
		T_PLC_MS := (DWORD_TO_UDINT(SHL(UDINT_TO_DWORD(T_PLC_MS),N) OR SHL(temp,N)) - UDINT#1) + Offset;
	END_IF;
END_FUNCTION_BLOCK

FUNCTION BIT_LOAD_DW:DWORD

	VAR_INPUT
		IN :	DWORD;
		VAL :	BOOL;
		POS :	INT;
	END_VAR

	IF val THEN
		BIT_LOAD_DW := in OR SHL(DWORD#1,pos);
	ELSE
		BIT_LOAD_DW := in AND (NOT SHL(DWORD#1,pos));
	END_IF;
END_FUNCTION

FUNCTION BIT_OF_DWORD : BOOL
  VAR_INPUT
    IN : DWORD;
    N : INT;
  END_VAR

  BIT_OF_DWORD := (SHR(in,N) AND 16#00000001) > 0;
  (* from OSCAT library; www.oscat.de  *)
END_FUNCTION

FUNCTION _INT_TO_UDINT:UDINT
	VAR_INPUT
		IN :	INT;
	END_VAR

	_INT_TO_UDINT := DINT_TO_UDINT(INT_TO_DINT(IN));
END_FUNCTION

FUNCTION _DWORD_TO_REAL:REAL
	VAR_INPUT
		IN :	DWORD;
	END_VAR

	_DWORD_TO_REAL := UDINT_TO_REAL(DWORD_TO_UDINT(IN));

END_FUNCTION

FUNCTION_BLOCK RDM_block
	VAR_INPUT
		LAST :	REAL;
	END_VAR
	VAR_OUTPUT
		RDM :	REAL;
	END_VAR
	VAR
		T_PLC_MS :	T_PLC_MS_block;
		tn :	DWORD;
		tc :	INT;
	END_VAR
	T_PLC_MS();
	tn := UDINT_TO_DWORD(T_PLC_MS.T_PLC_MS);
	tc := Bit_Count(tn);

	tn:=BIT_LOAD_DW(tn,BIT_OF_DWORD(tn,2),31); (* tn.31 := tn.2; *)
	tn:=BIT_LOAD_DW(tn,BIT_OF_DWORD(tn,5),30); (* tn.30 := tn.5; *)
	tn:=BIT_LOAD_DW(tn,BIT_OF_DWORD(tn,4),29); (* tn.29 := tn.4; *)
	tn:=BIT_LOAD_DW(tn,BIT_OF_DWORD(tn,1),28); (* tn.28 := tn.1; *)
	tn:=BIT_LOAD_DW(tn,BIT_OF_DWORD(tn,0),27); (* tn.27 := tn.0; *)
	tn:=BIT_LOAD_DW(tn,BIT_OF_DWORD(tn,7),26); (* tn.26 := tn.7; *)
	tn:=BIT_LOAD_DW(tn,BIT_OF_DWORD(tn,6),25); (* tn.25 := tn.6; *)
	tn:=BIT_LOAD_DW(tn,BIT_OF_DWORD(tn,3),24); (* tn.24 := tn.3; *)

	tn := ROL(tn,Bit_Count(tn)) OR DWORD#16#80000001;
	tn := UDINT_TO_DWORD(DWORD_TO_UDINT(tn) MOD UDINT#71474513 + _INT_TO_UDINT(tc) + UDINT#77);
	RDM := fract(_DWORD_TO_REAL(tn) / 10000000.0 * (2.71828182845904523536028747135266249 - LIMIT_REAL(0.0,last,1.0)));
END_FUNCTION_BLOCK

FUNCTION_BLOCK RDM22
	VAR_INPUT
		LAST :	INT;
		LOW :	INT;
		HIGH :	INT;
	END_VAR

	VAR_OUTPUT
		RDM2 :	INT;
	END_VAR

	VAR
		rdm :	RDM_block;
	END_VAR

	rdm(last:=fract(INT_TO_REAL(last) * 3.14159265358979323846264338327950288));
	RDM2 := TRUNC(rdm.RDM * INT_TO_REAL(high - low + 1)) + low;
END_FUNCTION_BLOCK

FUNCTION_BLOCK _ARRAY_SHUFFLE2
	VAR_IN_OUT
		PT :	oscat_pt_ARRAY;
	END_VAR

	VAR_INPUT
		SIZE :	UINT;
	END_VAR

	VAR_OUTPUT
		_ARRAY_SHUFFLE :	BOOL;
	END_VAR
	VAR
		temp :	REAL;
		pos :	INT;
		i :	INT;
		stop :	INT;
		rdm2 :	rdm22;
	END_VAR

	stop :=LIMIT_INT(1,UINT_TO_INT(size),1000);
	FOR i := 1 TO stop DO
			rdm2(last:=i+pos,low:=1,high:=stop);
			pos := rdm2.rdm2;
			(* swap elements *)
			temp := pt[i];
			pt[i] := pt[pos];
			pt[pos] := temp;
	END_FOR;

	_ARRAY_SHUFFLE := TRUE;
END_FUNCTION_BLOCK

PROGRAM program0
  VAR
    LocalVar0 : oscat_pt_ARRAY;
    LocalVar1 : UINT;
	LocalOUT  : BOOL;
	func_block : _ARRAY_SHUFFLE2;
  END_VAR
	func_block.pt := LocalVar0;
	func_block.size := LocalVar1;
	func_block();
	LocalOUT := func_block._ARRAY_SHUFFLE;

END_PROGRAM

CONFIGURATION Config0
	VAR_GLOBAL
		PLC_TICKS_PER_SEC :	INT;
		PLC_SYS_TICK_CNT :	DINT;
	END_VAR
  RESOURCE Res0 ON PLC
    TASK task0(INTERVAL := T#20ms,PRIORITY := 0);
    PROGRAM instance0 WITH task0 : program0;
  END_RESOURCE
END_CONFIGURATION

(* ---- _ARRAY_SORT.ST ---- *)
TYPE
	oscat_pt_ARRAY: ARRAY [1..100] OF REAL;
	oscat_stack_array: ARRAY [1..32]   OF INT;
END_TYPE

FUNCTION _INT_TO_UDINT:UDINT
	VAR_INPUT
		IN :	INT;
	END_VAR

	_INT_TO_UDINT := DINT_TO_UDINT(INT_TO_DINT(IN));
END_FUNCTION

FUNCTION_BLOCK _ARRAY_SORT2
	VAR_IN_OUT
		PT :	oscat_pt_ARRAY;
	END_VAR

	VAR_INPUT
		SIZE :	UINT;
	END_VAR

	VAR_OUTPUT
		_ARRAY_SORT :BOOL;
	END_VAR

	VAR
		stack_count :	INT;
		stack :	oscat_stack_array;
		links :	INT;
		rechts :	INT;
		pivot :	REAL;
		i :	INT;
		j :	INT;
		ende_innen :	BOOL;
		ende_aussen :	BOOL;
		tmp :	REAL;
		x :	INT;
	END_VAR

	links := 1;
	rechts := DWORD_TO_INT(SHR(UINT_TO_DWORD(size),2));
	stack_count := 1;

	WHILE NOT ende_aussen DO
		IF links < rechts THEN
			x := DWORD_TO_INT(SHR(UDINT_TO_DWORD(_INT_TO_UDINT(rechts)+ _INT_TO_UDINT(links)),1));
			pivot := PT[x];
			i := links - 1;
			j := rechts + 1;

			ende_innen := FALSE;
			REPEAT
				REPEAT	i := i+1;	UNTIL (PT[i] >= pivot) OR NOT (i < rechts)	END_REPEAT;
				REPEAT	j := j-1;	UNTIL (PT[j] <= pivot) OR NOT (j > links)	END_REPEAT;
				IF i >= j THEN
					ende_innen := TRUE;
				ELSE
					tmp := PT[j];
					PT[j] := PT[i];
					PT[i] := tmp;
				END_IF;

			UNTIL ende_innen END_REPEAT;

			stack[stack_count] := rechts;
			IF Stack_count < 32 THEN
				stack_count := stack_count +1;
			ELSE
				ende_aussen := TRUE;
				_ARRAY_SORT := FALSE;
			END_IF;
			rechts := MAX(links, i-1);

		ELSE
			IF stack_count = 1 THEN
				ende_aussen := TRUE;
			ELSE
				links := rechts+1;
				stack_count := stack_count - 1;
				rechts:= stack[stack_count];
			END_IF;
		END_IF;
	END_WHILE;

	_ARRAY_SORT := TRUE;
END_FUNCTION_BLOCK

PROGRAM program0
  VAR
    LocalVar0 : oscat_pt_ARRAY;
    LocalVar1 : UINT;
	LocalOUT  : BOOL;
	func_block : _ARRAY_SORT2;
  END_VAR
	func_block.pt := LocalVar0;
	func_block.size := LocalVar1;
	func_block();
	LocalOUT := func_block._ARRAY_SORT;

END_PROGRAM

CONFIGURATION Config0
  RESOURCE Res0 ON PLC
    TASK task0(INTERVAL := T#20ms,PRIORITY := 0);
    PROGRAM instance0 WITH task0 : program0;
  END_RESOURCE
END_CONFIGURATION

(* ---- _BUFFER_UPPERCASE_NW.ST ---- *)
TYPE
  oscat_NW_BUF_LONG  : ARRAY [0..4095] OF BYTE;
END_TYPE

FUNCTION SETUP_EXTENDED_ASCII:BOOL
	VAR_INPUT
		X :	BOOL;
	END_VAR

	SETUP_EXTENDED_ASCII := X OR TRUE;
END_FUNCTION

FUNCTION TO_UPPER:BYTE

	VAR_INPUT
		IN :	BYTE;
	END_VAR

	IF in > BYTE#96 AND in < BYTE#123 THEN
	TO_UPPER := in AND BYTE#16#DF;
	ELSIF in > BYTE#223 AND in <> BYTE#247 AND in <> BYTE#255 AND SETUP_EXTENDED_ASCII(FALSE) THEN
	TO_UPPER := in AND BYTE#16#DF;
	ELSE
	TO_UPPER := in;
	END_IF;

END_FUNCTION

FUNCTION_BLOCK _BUFFER_UPPERCASE_NW
	VAR_INPUT
		SIZE :	UINT;
	END_VAR

	VAR_OUTPUT
		_BUFFER_UPPERCASE :	BOOL;
	END_VAR

	VAR_IN_OUT
		PT :	oscat_NW_BUF_LONG;
	END_VAR

	VAR
		pos :	INT;
		size2 :	INT;
	END_VAR

	pos := 0;
	size2 := UINT_TO_INT(SIZE);

	WHILE pos < size2 DO
		PT[pos] := TO_UPPER(PT[pos]);
		pos := pos + 1;
	END_WHILE;

	_BUFFER_UPPERCASE := TRUE;

END_FUNCTION_BLOCK

PROGRAM program0
  VAR
	SIZE :	UINT;

	_BUFFER_UPPERCASE :	BOOL;

	PT :	oscat_NW_BUF_LONG;

	func_block : _BUFFER_UPPERCASE_NW;
  END_VAR
	func_block.SIZE  :=SIZE ;
	func_block.PT  :=PT ;
	func_block();
	PT := func_block.PT;
	_BUFFER_UPPERCASE := func_block._BUFFER_UPPERCASE;
END_PROGRAM

CONFIGURATION Config0
  RESOURCE Res0 ON PLC
    TASK task0(INTERVAL := T#20ms,PRIORITY := 0);
    PROGRAM instance0 WITH task0 : program0;
  END_RESOURCE
END_CONFIGURATION

(* ---- _INSERT80.ST ---- *)
FUNCTION_BLOCK _INSERT80

    VAR_INPUT
        IN1 :	STRING;
        IN2 :	STRING;
        P :	INT;
    END_VAR

    VAR_OUTPUT
        _INSERT :	STRING;
    END_VAR

    VAR
        size :	INT;
    END_VAR

    size := LEN(IN1);
    IF size + LEN(IN2) <= 80 THEN
        P := LIMIT(0,P,size);
        IF P = 0 THEN
            _INSERT := CONCAT(IN2,IN1);
        ELSE
            _INSERT := INSERT(IN1, IN2, P);
        END_IF;
    END_IF;

END_FUNCTION_BLOCK

PROGRAM program0
	VAR
	    LocalVar1 : STRING;
        LocalVar2 : STRING;
        LocalVar3 : INT;
		LocalOUT  : STRING;
		func_block : _INSERT80;
  	END_VAR
	func_block.IN1 := LocalVar1;
    func_block.IN2 := LocalVar2;
    func_block.P := LocalVar3;
	func_block();
	LocalOUT := func_block._INSERT;
END_PROGRAM

CONFIGURATION Config0
  	RESOURCE Res0 ON PLC
    	TASK task0(INTERVAL := T#20ms,PRIORITY := 0);
    	PROGRAM instance0 WITH task0 : program0;
  	END_RESOURCE
END_CONFIGURATION

(* ---- _RMP_B.ST ---- *)
FUNCTION UDINT_TO_TIME2:TIME

	VAR_INPUT
		IN :	UDINT;
	END_VAR

	UDINT_TO_TIME2 := DINT_TO_TIME(UDINT_TO_DINT(IN));

END_FUNCTION

FUNCTION_BLOCK T_PLC_MS_block
	VAR_OUTPUT
		T_PLC_MS :	UDINT;
	END_VAR

	VAR_EXTERNAL
		PLC_TICKS_PER_SEC :	INT;
		PLC_SYS_TICK_CNT :	DINT;
	END_VAR

	VAR
		debug :	BOOL;(*Debug-Mode ON / OFF*)
		N :	INT;(*Debug-Faktor*)
		Offset :	UDINT;(*Debug-Offset*)
		temp :	DWORD := DWORD#1;(*Debug-Offset*)
		mode :	BOOL;(*modus*)
		faktor :	UDINT;(*Systemtakt-Faktor*)
		init :	BOOL;
		v_plc_ticks_per_sec :	UDINT;
		base :	UDINT := UDINT#1000;
	END_VAR

	IF init = FALSE THEN
		v_plc_ticks_per_sec := INT_TO_UDINT(PLC_TICKS_PER_SEC);
		IF v_plc_ticks_per_sec = UDINT#1024 THEN
			faktor := UDINT#1;
			mode := FALSE;
		ELSIF v_plc_ticks_per_sec > UDINT#0 THEN
			IF v_plc_ticks_per_sec <= base THEN
				faktor := base / v_plc_ticks_per_sec;
				mode := FALSE;
			ELSE
				faktor := v_plc_ticks_per_sec / base;
				mode := TRUE;
			END_IF;
		ELSE
			faktor := UDINT#1;
		END_IF;
		init := TRUE;
	END_IF;

	IF mode THEN
		T_PLC_MS := DINT_TO_UDINT(PLC_SYS_TICK_CNT) / faktor;
	ELSE
		T_PLC_MS := DINT_TO_UDINT(PLC_SYS_TICK_CNT) * faktor;
	END_IF;

	IF debug THEN
		T_PLC_MS := (DWORD_TO_UDINT(SHL(UDINT_TO_DWORD(T_PLC_MS),N) OR SHL(temp,N)) - UDINT#1) + Offset;
	END_IF;

END_FUNCTION_BLOCK

FUNCTION TIME_TO_UDINT2:UDINT
	VAR_INPUT
		X :	TIME;
	END_VAR

	TIME_TO_UDINT2 := DINT_TO_UDINT(TIME_TO_DINT(X));
END_FUNCTION

FUNCTION FRMP_B:BYTE
	VAR_INPUT
		START :	BYTE;
		DIR :	BOOL;
		TD :	TIME;
		TR :	TIME;
	END_VAR

	IF TD < TR THEN
		FRMP_B := MIN(UDINT_TO_BYTE(DWORD_TO_UDINT(SHL(TIME_TO_DWORD(TD), 8)) / TIME_TO_UDINT2(TR)), SEL(DIR, START, USINT_TO_BYTE(USINT#255 - BYTE_TO_USINT(START))));
		IF DIR THEN
			FRMP_B := USINT_TO_BYTE(BYTE_TO_USINT(START) + BYTE_TO_USINT(FRMP_B));
		ELSE
			FRMP_B := USINT_TO_BYTE(BYTE_TO_USINT(START) - BYTE_TO_USINT(FRMP_B));
		END_IF;
	ELSE
		FRMP_B := SEL(DIR, BYTE#0, BYTE#255);
	END_IF;
END_FUNCTION

FUNCTION_BLOCK _RMP_B
	VAR_INPUT
		DIR :	BOOL;
		E :	BOOL := TRUE;
		TR :	TIME;
	END_VAR

	VAR_IN_OUT
		RMP :	BYTE;
	END_VAR

	VAR
		T_PLC_MS :	T_PLC_MS_block;
		tx :	TIME;
		tl :	TIME;
		tn :	TIME;
		init :	BOOL;
		last_dir :	BOOL;
		start :	BYTE;
	END_VAR

	T_PLC_MS();
	tx := UDINT_TO_TIME(T_PLC_MS.T_PLC_MS);

	IF E AND init AND (dir = last_dir) AND (RMP <> SEL(DIR, BYTE#0, BYTE#255)) AND TR = tn THEN
		RMP := FRMP_B(start, DIR, tx - tl, TR);
	ELSE
		init := TRUE;
		tl := tx;
		tn := tr;
		start := RMP;
	END_IF;
	last_dir := dir;
END_FUNCTION_BLOCK

PROGRAM program0
	VAR
	    LocalVar1 : BOOL;
		LocalVar2 : BOOL;
		LocalVar3 : TIME;
		LocalVar4 : BYTE;
		func_block : _RMP_B;
  	END_VAR
	func_block.DIR := LocalVar1;
	func_block.E := LocalVar2;
	func_block.TR := LocalVar3;
	func_block.RMP := LocalVar4;
	func_block();
	LocalVar4 := func_block.RMP;
END_PROGRAM

CONFIGURATION Config0
	VAR_GLOBAL
		PLC_TICKS_PER_SEC :	INT;
		PLC_SYS_TICK_CNT :	DINT;
	END_VAR
  	RESOURCE Res0 ON PLC
    	TASK task0(INTERVAL := T#20ms,PRIORITY := 0);
    	PROGRAM instance0 WITH task0 : program0;
  	END_RESOURCE
END_CONFIGURATION

(* ---- _RMP_NEXT.ST ---- *)
FUNCTION UDINT_TO_TIME2:TIME

	VAR_INPUT
		IN :	UDINT;
	END_VAR

	UDINT_TO_TIME2 := DINT_TO_TIME(UDINT_TO_DINT(IN));

END_FUNCTION

FUNCTION_BLOCK T_PLC_MS_block
	VAR_OUTPUT
		T_PLC_MS :	UDINT;
	END_VAR

	VAR_EXTERNAL
		PLC_TICKS_PER_SEC :	INT;
		PLC_SYS_TICK_CNT :	DINT;
	END_VAR

	VAR
		debug :	BOOL;(*Debug-Mode ON / OFF*)
		N :	INT;(*Debug-Faktor*)
		Offset :	UDINT;(*Debug-Offset*)
		temp :	DWORD := DWORD#1;(*Debug-Offset*)
		mode :	BOOL;(*modus*)
		faktor :	UDINT;(*Systemtakt-Faktor*)
		init :	BOOL;
		v_plc_ticks_per_sec :	UDINT;
		base :	UDINT := UDINT#1000;
	END_VAR

	IF init = FALSE THEN
		v_plc_ticks_per_sec := INT_TO_UDINT(PLC_TICKS_PER_SEC);
		IF v_plc_ticks_per_sec = UDINT#1024 THEN
			faktor := UDINT#1;
			mode := FALSE;
		ELSIF v_plc_ticks_per_sec > UDINT#0 THEN
			IF v_plc_ticks_per_sec <= base THEN
				faktor := base / v_plc_ticks_per_sec;
				mode := FALSE;
			ELSE
				faktor := v_plc_ticks_per_sec / base;
				mode := TRUE;
			END_IF;
		ELSE
			faktor := UDINT#1;
		END_IF;
		init := TRUE;
	END_IF;

	IF mode THEN
		T_PLC_MS := DINT_TO_UDINT(PLC_SYS_TICK_CNT) / faktor;
	ELSE
		T_PLC_MS := DINT_TO_UDINT(PLC_SYS_TICK_CNT) * faktor;
	END_IF;

	IF debug THEN
		T_PLC_MS := (DWORD_TO_UDINT(SHL(UDINT_TO_DWORD(T_PLC_MS),N) OR SHL(temp,N)) - UDINT#1) + Offset;
	END_IF;
END_FUNCTION_BLOCK

FUNCTION TIME_TO_UDINT2:UDINT
	VAR_INPUT
		X :	TIME;
	END_VAR

	TIME_TO_UDINT2 := DINT_TO_UDINT(TIME_TO_DINT(X));
END_FUNCTION

FUNCTION FRMP_B:BYTE
	VAR_INPUT
		START :	BYTE;
		DIR :	BOOL;
		TD :	TIME;
		TR :	TIME;
	END_VAR

	IF TD < TR THEN
		FRMP_B := MIN(UDINT_TO_BYTE(DWORD_TO_UDINT(SHL(TIME_TO_DWORD(TD), 8)) / TIME_TO_UDINT2(TR)), SEL(DIR, START, USINT_TO_BYTE(USINT#255 - BYTE_TO_USINT(START))));
		IF DIR THEN
			FRMP_B := USINT_TO_BYTE(BYTE_TO_USINT(START) + BYTE_TO_USINT(FRMP_B));
		ELSE
			FRMP_B := USINT_TO_BYTE(BYTE_TO_USINT(START) - BYTE_TO_USINT(FRMP_B));
		END_IF;
	ELSE
		FRMP_B := SEL(DIR, BYTE#0, BYTE#255);
	END_IF;
END_FUNCTION

FUNCTION_BLOCK _RMP_B
	VAR_INPUT
		DIR :	BOOL;
		E :	BOOL := TRUE;
		TR :	TIME;
	END_VAR

	VAR_IN_OUT
		RMP :	BYTE;
	END_VAR

	VAR
		T_PLC_MS :	T_PLC_MS_block;
		tx :	TIME;
		tl :	TIME;
		tn :	TIME;
		init :	BOOL;
		last_dir :	BOOL;
		start :	BYTE;
	END_VAR

	T_PLC_MS();
	tx := UDINT_TO_TIME(T_PLC_MS.T_PLC_MS);

	IF E AND init AND (dir = last_dir) AND (RMP <> SEL(DIR, BYTE#0, BYTE#255)) AND TR = tn THEN
		RMP := FRMP_B(start, DIR, tx - tl, TR);
	ELSE
		init := TRUE;
		tl := tx;
		tn := tr;
		start := RMP;
	END_IF;
	last_dir := dir;
END_FUNCTION_BLOCK

FUNCTION_BLOCK TREND_DW
	VAR_INPUT
		X :	DWORD;
	END_VAR
	VAR_OUTPUT
		Q :	BOOL;
		TU :	BOOL;
		TD :	BOOL;
		D :	DWORD;
	END_VAR

	VAR
		LAST_X :	DWORD;
	END_VAR

	IF X > last_X THEN
		TU := TRUE;
		TD := FALSE;
		D := UDINT_TO_DWORD(DWORD_TO_UDINT(X) - DWORD_TO_UDINT(last_X));
		Q := TRUE;
	ELSIF X < last_X THEN
		TD := TRUE;
		TU := FALSE;
		D := UDINT_TO_DWORD(DWORD_TO_UDINT(last_X) - DWORD_TO_UDINT(X));
		Q := FALSE;
	ELSE
		TU := FALSE;
		TD := FALSE;
		D := DWORD#0;
	END_IF;
	last_X := X;
END_FUNCTION_BLOCK

FUNCTION_BLOCK _RMP_NEXT
	VAR_INPUT
		E :	BOOL := TRUE;
		IN :	BYTE;
		TR :	TIME;
		TF :	TIME;
		TL :	TIME;
	END_VAR

	VAR_OUTPUT
		DIR :	BOOL;
		UP :	BOOL;
		DN :	BOOL;
	END_VAR

	VAR_IN_OUT
		OUT :	BYTE;
	END_VAR
	VAR
		rmx :	_RMP_B;
		dirx :	TREND_DW;
		t_lock :	TP;
		xen :	BOOL;
		xdir :	BOOL;
	END_VAR

	dirx(X := BYTE_TO_DWORD(in));

	t_lock(in := FALSE, pt := TL);

	IF dirx.TU AND (OUT < IN) THEN
		IF NOT xdir AND xen THEN t_lock(in := TRUE); END_IF;
		xen := TRUE;
		xdir := TRUE;
	ELSIF dirx.TD AND (OUT > IN) THEN
		IF xdir AND xen THEN t_lock(in := TRUE); END_IF;
		xen := TRUE;
		xdir := FALSE;
	ELSIF xen THEN
		IF (xdir AND (out >= in)) OR (NOT xdir AND (out <= in)) THEN
			xen := FALSE;
			IF tl > t#0s THEN t_lock(IN := TRUE); END_IF;
		END_IF;
	END_IF;

	IF NOT t_lock.Q AND xen THEN
		UP := XDIR;
		DIR := XDIR;
		DN := NOT XDIR;
	ELSE
		UP := FALSE;
		DN := FALSE;
	END_IF;

	rmx(rmp := OUT, E := E AND (UP OR DN) , dir := DIR, tr := SEL(dir, TF, TR));
	OUT := rmx.RMP;
END_FUNCTION_BLOCK

PROGRAM program0
	VAR
	    LocalVar1 : BOOL;
		LocalVar2 : BYTE;
		LocalVar3 : TIME;
		LocalVar4 : TIME;
		LocalVar5 : TIME;
		LocalVar6 : BOOL;
		LocalVar7 : BOOL;
		LocalVar8 : BOOL;
		LocalInOut : BYTE;
		func_block : _RMP_NEXT;
  	END_VAR
	func_block.E  := LocalVar1;
	func_block.IN := LocalVar2;
	func_block.TR := LocalVar3;
	func_block.TF := LocalVar4;
	func_block.TL := LocalVar5;
	func_block.OUT := LocalInOut;
	func_block();
	LocalInOut := func_block.OUT;
	LocalVar6 := func_block.DIR;
	LocalVar7 := func_block.UP;
	LocalVar8 := func_block.DN;
END_PROGRAM

CONFIGURATION Config0
	VAR_GLOBAL
		PLC_TICKS_PER_SEC :	INT;
		PLC_SYS_TICK_CNT :	DINT;
	END_VAR
  	RESOURCE Res0 ON PLC
    	TASK task0(INTERVAL := T#20ms,PRIORITY := 0);
    	PROGRAM instance0 WITH task0 : program0;
  	END_RESOURCE
END_CONFIGURATION

(* ---- _RMP_W.ST ---- *)
FUNCTION_BLOCK T_PLC_MS_block
	VAR_OUTPUT
		T_PLC_MS :	UDINT;
	END_VAR

	VAR_EXTERNAL
		PLC_TICKS_PER_SEC :	INT;
		PLC_SYS_TICK_CNT :	DINT;
	END_VAR

	VAR
		debug :	BOOL;(*Debug-Mode ON / OFF*)
		N :	INT;(*Debug-Faktor*)
		Offset :	UDINT;(*Debug-Offset*)
		temp :	DWORD := DWORD#1;(*Debug-Offset*)
		mode :	BOOL;(*modus*)
		faktor :	UDINT;(*Systemtakt-Faktor*)
		init :	BOOL;
		v_plc_ticks_per_sec :	UDINT;
		base :	UDINT := UDINT#1000;
	END_VAR

	IF init = FALSE THEN
		v_plc_ticks_per_sec := INT_TO_UDINT(PLC_TICKS_PER_SEC);
		IF v_plc_ticks_per_sec = UDINT#1024 THEN
			faktor := UDINT#1;
			mode := FALSE;
		ELSIF v_plc_ticks_per_sec > UDINT#0 THEN
			IF v_plc_ticks_per_sec <= base THEN
				faktor := base / v_plc_ticks_per_sec;
				mode := FALSE;
			ELSE
				faktor := v_plc_ticks_per_sec / base;
				mode := TRUE;
			END_IF;
		ELSE
			faktor := UDINT#1;
		END_IF;
		init := TRUE;
	END_IF;

	IF mode THEN
		T_PLC_MS := DINT_TO_UDINT(PLC_SYS_TICK_CNT) / faktor;
	ELSE
		T_PLC_MS := DINT_TO_UDINT(PLC_SYS_TICK_CNT) * faktor;
	END_IF;

	IF debug THEN
		T_PLC_MS := (DWORD_TO_UDINT(SHL(UDINT_TO_DWORD(T_PLC_MS),N) OR SHL(temp,N)) - UDINT#1) + Offset;
	END_IF;
END_FUNCTION_BLOCK

FUNCTION _WORD_TO_DINT:DINT
	VAR_INPUT
		IN :	WORD;
	END_VAR
	_WORD_TO_DINT := UINT_TO_DINT(WORD_TO_UINT(IN));
END_FUNCTION

FUNCTION TIME_TO_UDINT2:UDINT
	VAR_INPUT
		X :	TIME;
	END_VAR

	TIME_TO_UDINT2 := DINT_TO_UDINT(TIME_TO_DINT(X));
END_FUNCTION

FUNCTION_BLOCK _RMP_W

	VAR_INPUT
		DIR :	BOOL;
		E :	BOOL := TRUE;
		TR :	TIME;
	END_VAR

	VAR_IN_OUT
		RMP :	WORD;
	END_VAR

	VAR
		T_PLC_MS :	T_PLC_MS_block;
		tx :	UDINT;
		tl :	UDINT;
		ptesss :	DINT;
		init :	BOOL;
		last_dir :	BOOL;
	END_VAR

	T_PLC_MS();
	tx := T_PLC_MS.T_PLC_MS;
	IF E AND init THEN
		(* we need to set tl = tx when direction changes *)
		IF dir XOR last_dir THEN
			tl := tx;
			last_dir := dir;
		END_IF;
		(* check_elapsed time and calculate only if necessary *)
		IF tr > t#0s THEN
			ptesss := DWORD_TO_DINT(UDINT_TO_DWORD(DWORD_TO_UDINT(SHL(UDINT_TO_DWORD(tx-tl), 16)) / TIME_TO_UDINT2(TR)));
		ELSE
			ptesss := DINT#65535;
		END_IF;
		IF ptesss > DINT#0 THEN
			(* perform the ptesss on the ramp *)
			tl := tx;
			(* calculate the ptesss response *)
			IF NOT dir THEN ptesss := - ptesss; END_IF;
			rmp := DINT_TO_WORD(LIMIT(DINT#0, _WORD_TO_DINT(rmp) + ptesss, DINT#65535));
		END_IF;
	ELSE
		tl := tx;
		init := TRUE;
	END_IF;
END_FUNCTION_BLOCK

PROGRAM program0
  VAR
		DIR :	BOOL;
		E   :	BOOL;
		TR  :	TIME;

		RMP :	WORD;

	func_block : _RMP_W;
  END_VAR
	func_block.DIR:=DIR;
	func_block.E  :=E  ;
	func_block.TR :=TR ;
	func_block();
	RMP := func_block.RMP;
END_PROGRAM

CONFIGURATION Config0
	VAR_GLOBAL
		PLC_TICKS_PER_SEC :	INT;
		PLC_SYS_TICK_CNT :	DINT;
	END_VAR
  	RESOURCE Res0 ON PLC
    	TASK task0(INTERVAL := T#20ms,PRIORITY := 0);
    	PROGRAM instance0 WITH task0 : program0;
  	END_RESOURCE
END_CONFIGURATION

(* ---- A_TRIG.ST ---- *)
FUNCTION_BLOCK A_TRIG

	VAR_INPUT
		IN :	REAL;
		RES :	REAL;
	END_VAR

	VAR_OUTPUT
		Q :	BOOL;
		D :	REAL;
	END_VAR

	VAR
		last_in :	REAL;
	END_VAR

	D := IN - LAST_IN;
	IF ABS(D) >= res THEN
		Q := TRUE;
		last_in := IN;
	ELSE
		Q := FALSE;
	END_IF;

END_FUNCTION_BLOCK

PROGRAM program0
	VAR
	    LocalVar0 : REAL;
		LocalVar1 : REAL;
		LocalOUT1  : BOOL;
		LocalOUT2  : REAL;
		func_block : A_TRIG;
  	END_VAR
	func_block.IN := LocalVar0;
    func_block.RES := LocalVar1;
	func_block();
	LocalOUT1 := func_block.Q;
	LocalOUT2 := func_block.D;
END_PROGRAM

CONFIGURATION Config0
  	RESOURCE Res0 ON PLC
    	TASK task0(INTERVAL := T#20ms,PRIORITY := 0);
    	PROGRAM instance0 WITH task0 : program0;
  	END_RESOURCE
END_CONFIGURATION

(* ---- ACTUATOR_3P.ST ---- *)
FUNCTION UDINT_TO_TIME2:TIME

	VAR_INPUT
		IN :	UDINT;
	END_VAR

	UDINT_TO_TIME2 := DINT_TO_TIME(UDINT_TO_DINT(IN));

END_FUNCTION

FUNCTION_BLOCK T_PLC_MS_block
	VAR_OUTPUT
		T_PLC_MS :	UDINT;
	END_VAR

	VAR_EXTERNAL
		PLC_TICKS_PER_SEC :	INT;
		PLC_SYS_TICK_CNT :	DINT;
	END_VAR

	VAR
		debug :	BOOL;(*Debug-Mode ON / OFF*)
		N :	INT;(*Debug-Faktor*)
		Offset :	UDINT;(*Debug-Offset*)
		temp :	DWORD := DWORD#1;(*Debug-Offset*)
		mode :	BOOL;(*modus*)
		faktor :	UDINT;(*Systemtakt-Faktor*)
		init :	BOOL;
		v_plc_ticks_per_sec :	UDINT;
		base :	UDINT := UDINT#1000;
	END_VAR

	IF init = FALSE THEN
		v_plc_ticks_per_sec := INT_TO_UDINT(PLC_TICKS_PER_SEC);
		IF v_plc_ticks_per_sec = UDINT#1024 THEN
			faktor := UDINT#1;
			mode := FALSE;
		ELSIF v_plc_ticks_per_sec > UDINT#0 THEN
			IF v_plc_ticks_per_sec <= base THEN
				faktor := base / v_plc_ticks_per_sec;
				mode := FALSE;
			ELSE
				faktor := v_plc_ticks_per_sec / base;
				mode := TRUE;
			END_IF;
		ELSE
			faktor := UDINT#1;
		END_IF;
		init := TRUE;
	END_IF;

	IF mode THEN
		T_PLC_MS := DINT_TO_UDINT(PLC_SYS_TICK_CNT) / faktor;
	ELSE
		T_PLC_MS := DINT_TO_UDINT(PLC_SYS_TICK_CNT) * faktor;
	END_IF;

	IF debug THEN
		T_PLC_MS := (DWORD_TO_UDINT(SHL(UDINT_TO_DWORD(T_PLC_MS),N) OR SHL(temp,N)) - UDINT#1) + Offset;
	END_IF;
END_FUNCTION_BLOCK

FUNCTION TIME_TO_UDINT2:UDINT
	VAR_INPUT
		X :	TIME;
	END_VAR

	TIME_TO_UDINT2 := DINT_TO_UDINT(TIME_TO_DINT(X));
END_FUNCTION

FUNCTION FRMP_B:BYTE
	VAR_INPUT
		START :	BYTE;
		DIR :	BOOL;
		TD :	TIME;
		TR :	TIME;
	END_VAR

	IF TD < TR THEN
		FRMP_B := MIN(UDINT_TO_BYTE(DWORD_TO_UDINT(SHL(TIME_TO_DWORD(TD), 8)) / TIME_TO_UDINT2(TR)), SEL(DIR, START, USINT_TO_BYTE(USINT#255 - BYTE_TO_USINT(START))));
		IF DIR THEN
			FRMP_B := USINT_TO_BYTE(BYTE_TO_USINT(START) + BYTE_TO_USINT(FRMP_B));
		ELSE
			FRMP_B := USINT_TO_BYTE(BYTE_TO_USINT(START) - BYTE_TO_USINT(FRMP_B));
		END_IF;
	ELSE
		FRMP_B := SEL(DIR, BYTE#0, BYTE#255);
	END_IF;
END_FUNCTION

FUNCTION_BLOCK _RMP_B
	VAR_INPUT
		DIR :	BOOL;
		E :	BOOL := TRUE;
		TR :	TIME;
	END_VAR

	VAR_IN_OUT
		RMP :	BYTE;
	END_VAR

	VAR
		T_PLC_MS :	T_PLC_MS_block;
		tx :	TIME;
		tl :	TIME;
		tn :	TIME;
		init :	BOOL;
		last_dir :	BOOL;
		start :	BYTE;
	END_VAR

	T_PLC_MS();
	tx := UDINT_TO_TIME(T_PLC_MS.T_PLC_MS);

	IF E AND init AND (dir = last_dir) AND (RMP <> SEL(DIR, BYTE#0, BYTE#255)) AND TR = tn THEN
		RMP := FRMP_B(start, DIR, tx - tl, TR);
	ELSE
		init := TRUE;
		tl := tx;
		tn := tr;
		start := RMP;
	END_IF;
	last_dir := dir;
END_FUNCTION_BLOCK

FUNCTION_BLOCK TREND_DW
	VAR_INPUT
		X :	DWORD;
	END_VAR
	VAR_OUTPUT
		Q :	BOOL;
		TU :	BOOL;
		TD :	BOOL;
		D :	DWORD;
	END_VAR

	VAR
		LAST_X :	DWORD;
	END_VAR

	IF X > last_X THEN
		TU := TRUE;
		TD := FALSE;
		D := UDINT_TO_DWORD(DWORD_TO_UDINT(X) - DWORD_TO_UDINT(last_X));
		Q := TRUE;
	ELSIF X < last_X THEN
		TD := TRUE;
		TU := FALSE;
		D := UDINT_TO_DWORD(DWORD_TO_UDINT(last_X) - DWORD_TO_UDINT(X));
		Q := FALSE;
	ELSE
		TU := FALSE;
		TD := FALSE;
		D := DWORD#0;
	END_IF;
	last_X := X;
END_FUNCTION_BLOCK

FUNCTION_BLOCK _RMP_NEXT_Block
	VAR_INPUT
		E :	BOOL := TRUE;
		IN :	BYTE;
		TR :	TIME;
		TF :	TIME;
		TL :	TIME;
	END_VAR

	VAR_OUTPUT
		DIR :	BOOL;
		UP :	BOOL;
		DN :	BOOL;
	END_VAR

	VAR_IN_OUT
		OUT :	BYTE;
	END_VAR
	VAR
		rmx :	_RMP_B;
		dirx :	TREND_DW;
		t_lock :	TP;
		xen :	BOOL;
		xdir :	BOOL;
	END_VAR

	dirx(X := BYTE_TO_DWORD(in));

	t_lock(in := FALSE, pt := TL);

	IF dirx.TU AND (OUT < IN) THEN
		IF NOT xdir AND xen THEN t_lock(in := TRUE); END_IF;
		xen := TRUE;
		xdir := TRUE;
	ELSIF dirx.TD AND (OUT > IN) THEN
		IF xdir AND xen THEN t_lock(in := TRUE); END_IF;
		xen := TRUE;
		xdir := FALSE;
	ELSIF xen THEN
		IF (xdir AND (out >= in)) OR (NOT xdir AND (out <= in)) THEN
			xen := FALSE;
			IF tl > t#0s THEN t_lock(IN := TRUE); END_IF;
		END_IF;
	END_IF;

	IF NOT t_lock.Q AND xen THEN
		UP := XDIR;
		DIR := XDIR;
		DN := NOT XDIR;
	ELSE
		UP := FALSE;
		DN := FALSE;
	END_IF;

	rmx(rmp := OUT, E := E AND (UP OR DN) , dir := DIR, tr := SEL(dir, TF, TR));
	OUT := rmx.RMP;
END_FUNCTION_BLOCK

FUNCTION _BYTE_TO_INT:INT
	VAR_INPUT
		IN :	BYTE;
	END_VAR

	_BYTE_TO_INT := USINT_TO_INT(BYTE_TO_USINT(IN));
END_FUNCTION

FUNCTION_BLOCK ACTUATOR_3P_Block

	VAR_INPUT
		IN :	BYTE;
		TEST :	BOOL;
		ARE :	BOOL := TRUE;
		END_POS :	BOOL;
		T_RUN :	TIME := T#60s;
		T_EXT :	TIME := T#10s;
		T_CAL :	TIME := T#600s;
		T_DIAG :	TIME := T#10d;
		SWITCH_AVAIL :	BOOL;
	END_VAR

	VAR_OUTPUT
		OUT1 :	BOOL;
		OUT2 :	BOOL;
		POS :	BYTE;
		ERROR :	BOOL;
		STATUS :	BYTE;
	END_VAR

	VAR_IN_OUT
		ARX :	BOOL;
	END_VAR

	VAR
		tx :	TIME;
		_ramp :	_RMP_NEXT_Block;
		next_cal :	TIME;
		next_diag :	TIME;
		last :	TIME;
		start :	TIME;
		T_PLC_MS :	T_PLC_MS_Block;
	END_VAR

	T_PLC_MS();
	tx := UDINT_TO_TIME(T_PLC_MS.T_PLC_MS);

	IF TEST THEN
		status := BYTE#103;
		start := tx;
		ARX := TRUE;
	END_IF;

	CASE _BYTE_TO_INT(status) OF
		0:
			IF ARE AND NOT ARX THEN
				status := BYTE#103;
				start := tx;
				ARX := TRUE;
			END_IF;

		100:
			IF T_DIAG > T#0s AND tx > next_diag AND ARE AND NOT ARX THEN
					status := BYTE#103;
					start := tx;
					ARX := TRUE;

			ELSIF T_CAL > T#0s AND tx > next_cal AND ARE AND NOT ARX THEN
				IF pos > BYTE#127 THEN
					OUT1 := TRUE;
					OUT2 := FALSE;
					_ramp.IN := BYTE#255;
					ARX := TRUE;
				ELSE
					OUT1 := FALSE;
					OUT2 := TRUE;
					_ramp.IN := BYTE#0;
					ARX := TRUE;
				END_IF;
				status := BYTE#101;
				start := tx;
			ELSE
				IF NOT(OUT1 OR OUT2) THEN next_cal := next_cal + (tx-last); END_IF;
				_ramp.IN := IN;
			END_IF;

		101:
			IF tx - start < T_EXT THEN
				next_cal := tx + T_CAL;
			ELSIF SWITCH_AVAIL AND END_POS THEN
				STATUS := BYTE#100;
				ARX := FALSE;
			ELSIF tx - start > T_EXT + T_RUN THEN
				ERROR := SWITCH_AVAIL;
				ARX := FALSE;
			END_IF;

		103:
			IF tx - start < T_EXT THEN
				ERROR := FALSE;
				_ramp.TR := T_RUN;
				_ramp.TF := T_RUN;
				OUT1 := TRUE;
				OUT2 := FALSE;
				_ramp.IN := BYTE#255;
			ELSIF SWITCH_AVAIL AND END_POS THEN
				_ramp.TR := tx - start;
				STATUS := BYTE#104;
			ELSIF tx - start > T_EXT + T_RUN THEN
				ERROR := SWITCH_AVAIL;
				STATUS := BYTE#104;
				start := tx;
			END_IF;

		104:
			IF tx - start < T_ext THEN
				OUT1 := FALSE;
				OUT2 := TRUE;
				_ramp.IN := BYTE#0;
				next_diag := tx + T_DIAG;
			ELSIF SWITCH_AVAIL AND END_POS THEN
				_ramp.TR := tx - start;
				IF DINT_TO_TIME(ABS(TIME_TO_DINT(_ramp.TR) - TIME_TO_DINT(_ramp.TF)) * DINT#10) > T_RUN THEN error := TRUE; END_IF;
				STATUS := BYTE#100;
				ARX := FALSE;
				next_cal := tx + T_CAL;
			ELSIF tx - start > T_EXT + T_RUN THEN
				IF SWITCH_AVAIL THEN ERROR := TRUE; END_IF;
				STATUS := BYTE#100;
				ARX := FALSE;
				next_CAL := tx + T_CAL;
			END_IF;
	END_CASE;

	_ramp(OUT := POS);
	POS := _ramp.OUT;
	IF STATUS = BYTE#100 THEN
		OUT1 := _ramp.UP;
		OUT2 := _ramp.DN;
	END_IF;

	IF SWITCH_AVAIL AND END_POS THEN
		POS := SEL_BYTE(POS > BYTE#127, BYTE#0, BYTE#255);
		next_cal := tx + T_CAL;
	END_IF;

	last := tx;

END_FUNCTION_BLOCK

PROGRAM program0
	VAR
		IN :	BYTE;
		TEST :	BOOL;
		ARE :	BOOL := TRUE;
		END_POS :	BOOL;
		T_RUN :	TIME := T#60s;
		T_EXT :	TIME := T#10s;
		T_CAL :	TIME := T#600s;
		T_DIAG :	TIME := T#10d;
		SWITCH_AVAIL :	BOOL;
		OUT1 :	BOOL;
		OUT2 :	BOOL;
		POS :	BYTE;
		ERROR :	BOOL;
		STATUS :	BYTE;
		func_block : ACTUATOR_3P_Block;
	END_VAR
	func_block.IN := IN;
	func_block.TEST := TEST;
	func_block.ARE := ARE ;
	func_block.END_POS := END_POS;
	func_block.T_RUN := T_RUN;
	func_block.T_EXT := T_EXT;
	func_block.T_CAL := T_CAL ;
	func_block.T_DIAG := T_DIAG;
	func_block.SWITCH_AVAIL := SWITCH_AVAIL;
	func_block();
	OUT1  := func_block.OUT1;
	OUT2  := func_block.OUT2;
	POS  := func_block.POS;
	ERROR  := func_block.ERROR;
	STATUS  := func_block.STATUS;
END_PROGRAM

CONFIGURATION Config0
	VAR_GLOBAL
		PLC_TICKS_PER_SEC :	INT;
		PLC_SYS_TICK_CNT :	DINT;
	END_VAR
  	RESOURCE Res0 ON PLC
    	TASK task0(INTERVAL := T#20ms,PRIORITY := 0);
    	PROGRAM instance0 WITH task0 : program0;
  	END_RESOURCE
END_CONFIGURATION

(* ---- ACTUATOR_A.ST ---- *)
FUNCTION_BLOCK T_PLC_MS_block
	VAR_OUTPUT
		T_PLC_MS :	UDINT;
	END_VAR

	VAR_EXTERNAL
		PLC_TICKS_PER_SEC :	INT;
		PLC_SYS_TICK_CNT :	DINT;
	END_VAR

	VAR
		debug :	BOOL;(*Debug-Mode ON / OFF*)
		N :	INT;(*Debug-Faktor*)
		Offset :	UDINT;(*Debug-Offset*)
		temp :	DWORD := DWORD#1;(*Debug-Offset*)
		mode :	BOOL;(*modus*)
		faktor :	UDINT;(*Systemtakt-Faktor*)
		init :	BOOL;
		v_plc_ticks_per_sec :	UDINT;
		base :	UDINT := UDINT#1000;
	END_VAR

	IF init = FALSE THEN
		v_plc_ticks_per_sec := INT_TO_UDINT(PLC_TICKS_PER_SEC);
		IF v_plc_ticks_per_sec = UDINT#1024 THEN
			faktor := UDINT#1;
			mode := FALSE;
		ELSIF v_plc_ticks_per_sec > UDINT#0 THEN
			IF v_plc_ticks_per_sec <= base THEN
				faktor := base / v_plc_ticks_per_sec;
				mode := FALSE;
			ELSE
				faktor := v_plc_ticks_per_sec / base;
				mode := TRUE;
			END_IF;
		ELSE
			faktor := UDINT#1;
		END_IF;
		init := TRUE;
	END_IF;

	IF mode THEN
		T_PLC_MS := DINT_TO_UDINT(PLC_SYS_TICK_CNT) / faktor;
	ELSE
		T_PLC_MS := DINT_TO_UDINT(PLC_SYS_TICK_CNT) * faktor;
	END_IF;

	IF debug THEN
		T_PLC_MS := (DWORD_TO_UDINT(SHL(UDINT_TO_DWORD(T_PLC_MS),N) OR SHL(temp,N)) - UDINT#1) + Offset;
	END_IF;

END_FUNCTION_BLOCK

FUNCTION_BLOCK CYCLE_4

	VAR_INPUT
		E :	BOOL := TRUE;
		T0 :	TIME;
		T1 :	TIME;
		T2 :	TIME;
		T3 :	TIME;
		S0 :	BOOL;
		SX :	INT;
		SL :	BOOL;
	END_VAR

	VAR_OUTPUT
		STATE :	INT;
	END_VAR

	VAR
		tx :	TIME;
		last :	TIME;
		init :	BOOL;
		T_PLC_MS :	T_PLC_MS_block;
	END_VAR

	T_PLC_MS();
	tx:= UDINT_TO_TIME(T_PLC_MS.T_PLC_MS);

	(* init on first cycle *)
	IF NOT init THEN
		init := TRUE;
		last := tx;
	END_IF;

	IF E THEN
		IF SL THEN
			(* when sx > 0 then the state sx is forced to start *)
			state:= LIMIT(0,SX,3);
			last := tx;
			(* this is to avoid to reset sx from the calling programm it does work fine on codesys but i am not sure about other systems, because we are writing to an input *)
			SL := FALSE;
		ELSE
			CASE state OF
				0 :	(* wait for T0 and switch to next cycle *)
					IF tx - last >= T0 THEN
						state := 1;
						last := tx;
					END_IF;
				1 : (* wait for T1 over 1st cycle *)
					IF tx - last >= T1 THEN
						state := 2;
						last := tx;
					END_IF;
				2 : (* wait for T1 over 1st cycle *)
					IF tx - last >= T2 THEN
						state := 3;
						last := tx;
					END_IF;
				3 : (* wait for T2 over 2nd cycle *)
					IF tx - last >= T3 THEN
						IF S0 THEN State := 0; END_IF; (* if S0 is false, the sequence stops at state 3 *)
						last := tx;
					END_IF;
			END_CASE;
		END_IF;
	ELSE
		state := 0;
		last := tx;
	END_IF;

END_FUNCTION_BLOCK

FUNCTION_BLOCK ACTUATOR_A_Block

	VAR_INPUT
		I1 :	BYTE;
		IS :	BOOL;
		I2 :	BYTE;
		RV :	BOOL;
		DX :	BOOL;
		RUNTIME :	TIME;
		SELF_ACT_TIME :	TIME;
		OUT_MIN :	DWORD;
		OUT_MAX :	DWORD;
	END_VAR

	VAR_OUTPUT
		Y :	DWORD;
	END_VAR

	VAR
		timer :	CYCLE_4;
		dx_edge :	BOOL;
	END_VAR

	timer(T0 := RUNTIME, T1 := RUNTIME, T3 := SELF_ACT_TIME, sl := DX AND NOT dx_edge, sx := 0, S0 := SELF_ACT_TIME > t#0s);
	dx_edge := dx;

	CASE timer.STATE OF
		0:
			Y := OUT_MIN;
		1:
			Y := OUT_MAX;
		3:
			IF rv THEN
				Y := UDINT_TO_DWORD(DWORD_TO_UDINT(OUT_MAX) - (DWORD_TO_UDINT(OUT_MAX) - DWORD_TO_UDINT(OUT_MIN)) * BYTE_TO_UDINT(SEL(IS, I1, I2)) / UDINT#255);
			ELSE
				Y := UDINT_TO_DWORD((DWORD_TO_UDINT(OUT_MAX) - DWORD_TO_UDINT(OUT_MIN)) * BYTE_TO_UDINT(SEL(IS, I1, I2)) / UDINT#255 + DWORD_TO_UDINT(OUT_MIN));
			END_IF;
	END_CASE;

END_FUNCTION_BLOCK

PROGRAM program0
	VAR
		I1 :	BYTE;
		IS :	BOOL;
		I2 :	BYTE;
		RV :	BOOL;
		DX :	BOOL;
		RUNTIME :	TIME;
		SELF_ACT_TIME :	TIME;
		OUT_MIN :	DWORD;
		OUT_MAX :	DWORD;
		Y :	DWORD;
		func_block : ACTUATOR_A_Block;
	END_VAR
	func_block.I1 := I1;
	func_block.IS := IS;
	func_block.I2 := I2 ;
	func_block.RV := RV;
	func_block.DX := DX;
	func_block.RUNTIME := RUNTIME;
	func_block.SELF_ACT_TIME := SELF_ACT_TIME ;
	func_block.OUT_MIN := OUT_MIN;
	func_block.OUT_MAX := OUT_MAX;
	func_block();
	Y  := func_block.Y;
END_PROGRAM

CONFIGURATION Config0
	VAR_GLOBAL
		PLC_TICKS_PER_SEC :	INT;
		PLC_SYS_TICK_CNT :	DINT;
	END_VAR
  	RESOURCE Res0 ON PLC
    	TASK task0(INTERVAL := T#20ms,PRIORITY := 0);
    	PROGRAM instance0 WITH task0 : program0;
  	END_RESOURCE
END_CONFIGURATION

(* ---- ACTUATOR_COIL.ST ---- *)
FUNCTION UDINT_TO_TIME2:TIME

	VAR_INPUT
		IN :	UDINT;
	END_VAR

	UDINT_TO_TIME2 := DINT_TO_TIME(UDINT_TO_DINT(IN));

END_FUNCTION

FUNCTION_BLOCK T_PLC_MS_block
	VAR_OUTPUT
		T_PLC_MS :	UDINT;
	END_VAR

	VAR_EXTERNAL
		PLC_TICKS_PER_SEC :	INT;
		PLC_SYS_TICK_CNT :	DINT;
	END_VAR

	VAR
		debug :	BOOL;(*Debug-Mode ON / OFF*)
		N :	INT;(*Debug-Faktor*)
		Offset :	UDINT;(*Debug-Offset*)
		temp :	DWORD := DWORD#1;(*Debug-Offset*)
		mode :	BOOL;(*modus*)
		faktor :	UDINT;(*Systemtakt-Faktor*)
		init :	BOOL;
		v_plc_ticks_per_sec :	UDINT;
		base :	UDINT := UDINT#1000;
	END_VAR

	IF init = FALSE THEN
		v_plc_ticks_per_sec := INT_TO_UDINT(PLC_TICKS_PER_SEC);
		IF v_plc_ticks_per_sec = UDINT#1024 THEN
			faktor := UDINT#1;
			mode := FALSE;
		ELSIF v_plc_ticks_per_sec > UDINT#0 THEN
			IF v_plc_ticks_per_sec <= base THEN
				faktor := base / v_plc_ticks_per_sec;
				mode := FALSE;
			ELSE
				faktor := v_plc_ticks_per_sec / base;
				mode := TRUE;
			END_IF;
		ELSE
			faktor := UDINT#1;
		END_IF;
		init := TRUE;
	END_IF;

	IF mode THEN
		T_PLC_MS := DINT_TO_UDINT(PLC_SYS_TICK_CNT) / faktor;
	ELSE
		T_PLC_MS := DINT_TO_UDINT(PLC_SYS_TICK_CNT) * faktor;
	END_IF;

	IF debug THEN
		T_PLC_MS := (DWORD_TO_UDINT(SHL(UDINT_TO_DWORD(T_PLC_MS),N) OR SHL(temp,N)) - UDINT#1) + Offset;
	END_IF;
END_FUNCTION_BLOCK

FUNCTION TIME_TO_UDINT2:UDINT
	VAR_INPUT
		X :	TIME;
	END_VAR

	TIME_TO_UDINT2 := DINT_TO_UDINT(TIME_TO_DINT(X));
END_FUNCTION

FUNCTION_BLOCK ACTUATOR_COIL_Block

	VAR_INPUT
		IN :	BOOL;
		SELF_ACT_CYCLE :	TIME := T#10d;
		SELF_ACT_TIME :	TIME := T#1s;
	END_VAR

	VAR_OUTPUT
		OUT :	BOOL;
		STATUS :	BYTE;
	END_VAR

	VAR
		last :	UDINT;
		init :	BOOL;
		tx :	UDINT;
		now :	UDINT;
		T_PLC_MS :	T_PLC_MS_Block;
	END_VAR

	T_PLC_MS();
	now := T_PLC_MS.T_PLC_MS;

	IF NOT init THEN
		last := now;
		init := TRUE;
	ELSIF IN THEN
		OUT := TRUE;
		STATUS := BYTE#101;
		LAST := now;
	ELSE
		OUT := FALSE;
		STATUS := BYTE#100;
		tx := now - last;
		IF (self_act_cycle > T#0s) AND (tx >= TIME_TO_UDINT2(self_act_cycle)) THEN
			OUT := TRUE;
			STATUS := BYTE#102;
			IF tx >= TIME_TO_UDINT2(self_act_cycle + self_act_time) THEN
				last := now;
				OUT := FALSE;
				STATUS := BYTE#100;
			END_IF;
		END_IF;
	END_IF;

END_FUNCTION_BLOCK

PROGRAM program0
	VAR
		IN :	BOOL;
		SELF_ACT_CYCLE :	TIME := T#10d;
		SELF_ACT_TIME :	TIME := T#1s;
		OUT :	BOOL;
		STATUS :	BYTE;
		func_block : ACTUATOR_COIL_Block;
	END_VAR
	func_block.IN := IN;
	func_block.SELF_ACT_CYCLE := SELF_ACT_CYCLE;
	func_block.SELF_ACT_TIME := SELF_ACT_TIME ;
	func_block();
	OUT  := func_block.OUT;
	STATUS  := func_block.STATUS;
END_PROGRAM

CONFIGURATION Config0
	VAR_GLOBAL
		PLC_TICKS_PER_SEC :	INT;
		PLC_SYS_TICK_CNT :	DINT;
	END_VAR
  	RESOURCE Res0 ON PLC
    	TASK task0(INTERVAL := T#20ms,PRIORITY := 0);
    	PROGRAM instance0 WITH task0 : program0;
  	END_RESOURCE
END_CONFIGURATION

(* ---- ACTUATOR_PUMP.ST ---- *)
FUNCTION_BLOCK T_PLC_MS_block
	VAR_OUTPUT
		T_PLC_MS :	UDINT;
	END_VAR

	VAR_EXTERNAL
		PLC_TICKS_PER_SEC :	INT;
		PLC_SYS_TICK_CNT :	DINT;
	END_VAR

	VAR
		debug :	BOOL;(*Debug-Mode ON / OFF*)
		N :	INT;(*Debug-Faktor*)
		Offset :	UDINT;(*Debug-Offset*)
		temp :	DWORD := DWORD#1;(*Debug-Offset*)
		mode :	BOOL;(*modus*)
		faktor :	UDINT;(*Systemtakt-Faktor*)
		init :	BOOL;
		v_plc_ticks_per_sec :	UDINT;
		base :	UDINT := UDINT#1000;
	END_VAR

	IF init = FALSE THEN
		v_plc_ticks_per_sec := INT_TO_UDINT(PLC_TICKS_PER_SEC);
		IF v_plc_ticks_per_sec = UDINT#1024 THEN
			faktor := UDINT#1;
			mode := FALSE;
		ELSIF v_plc_ticks_per_sec > UDINT#0 THEN
			IF v_plc_ticks_per_sec <= base THEN
				faktor := base / v_plc_ticks_per_sec;
				mode := FALSE;
			ELSE
				faktor := v_plc_ticks_per_sec / base;
				mode := TRUE;
			END_IF;
		ELSE
			faktor := UDINT#1;
		END_IF;
		init := TRUE;
	END_IF;

	IF mode THEN
		T_PLC_MS := DINT_TO_UDINT(PLC_SYS_TICK_CNT) / faktor;
	ELSE
		T_PLC_MS := DINT_TO_UDINT(PLC_SYS_TICK_CNT) * faktor;
	END_IF;

	IF debug THEN
		T_PLC_MS := (DWORD_TO_UDINT(SHL(UDINT_TO_DWORD(T_PLC_MS),N) OR SHL(temp,N)) - UDINT#1) + Offset;
	END_IF;

END_FUNCTION_BLOCK

FUNCTION_BLOCK ONTIME_Block

	VAR_INPUT
		IN :	BOOL;
		RST :	BOOL;
	END_VAR

	VAR_IN_OUT
		SECONDS :	UDINT;
		CYCLES :	UDINT;
	END_VAR

	VAR
		tx :	UDINT;
		last :	UDINT;
		edge :	BOOL;
		init :	BOOL;
		ms :	UDINT;
		T_PLC_MS :	T_PLC_MS_Block;
	END_VAR

	T_PLC_MS();
	tx:= T_PLC_MS.T_PLC_MS;

	IF NOT init THEN
		init := TRUE;
		last := tx;
		ms := UDINT#0;
	END_IF;
	IF RST THEN
		SECONDS := UDINT#0;
		CYCLES := UDINT#0;
		last := tx;
		ms := UDINT#0;
	ELSIF IN THEN
		(* add the current milliseconds *)
		ms := (tx - last) + ms;
		IF ms >= UDINT#1000 THEN
			seconds := seconds + UDINT#1;
			ms := ms - UDINT#1000;
		END_IF;
		cycles := cycles + BOOL_TO_UDINT(NOT edge);
	END_IF;
	last := tx;
	edge := in;

END_FUNCTION_BLOCK

FUNCTION_BLOCK ACTUATOR_PUMP_Block

	VAR_INPUT
		IN :	BOOL;
		MANUAL :	BOOL;
		RST :	BOOL := FALSE;
		MIN_ONTIME :	TIME := T#10s;
		MIN_OFFTIME :	TIME := T#10s;
		RUN_EVERY :	TIME := T#10000m;
	END_VAR

	VAR_OUTPUT
		PUMP :	BOOL;
		RUNTIME :	UDINT;
		CYCLES :	UDINT;
	END_VAR

	VAR
		tx :	TIME;
		last_change :	TIME;
		meter :	ONTIME_Block;
		old_man :	BOOL;
		init :	BOOL;
		T_PLC_MS :	T_PLC_MS_Block;
	END_VAR

	T_PLC_MS();
	tx:= UDINT_TO_TIME(T_PLC_MS.T_PLC_MS);

	IF NOT init THEN
		init := TRUE;
		last_change := tx;
	ELSIF rst THEN
		rst := FALSE;
		runtime := UDINT#0;
		cycles := UDINT#0;
	ELSIF manual AND NOT pump AND NOT old_man THEN
		last_change := tx;
		pump := TRUE;
	ELSIF NOT manual AND old_man AND pump AND NOT in THEN
		last_change := tx;
		pump := FALSE;
	ELSIF in AND NOT pump AND tx - last_change >= min_offtime THEN
		last_change := tx;
		pump := TRUE;
	ELSIF pump AND NOT in AND NOT manual AND tx - last_change >= min_ontime THEN
		last_change := tx;
		pump := FALSE;
	ELSIF NOT pump AND (tx - last_change >= run_every) AND (run_every > T#0s) THEN
		last_change := tx;
		pump := TRUE;
	END_IF;

	meter(in := pump, SECONDS := runtime, CYCLES := cycles);
	cycles := meter.CYCLES;
	runtime := meter.SECONDS;

	old_man := manual;

END_FUNCTION_BLOCK

PROGRAM program0
	VAR
		IN :	BOOL;
		MANUAL :	BOOL;
		RST :	BOOL := FALSE;
		MIN_ONTIME :	TIME := T#10s;
		MIN_OFFTIME :	TIME := T#10s;
		RUN_EVERY :	TIME := T#10000m;
		PUMP :	BOOL;
		RUNTIME :	UDINT;
		CYCLES :	UDINT;
		func_block : ACTUATOR_PUMP_Block;
	END_VAR
	func_block.IN := IN;
	func_block.MANUAL := MANUAL;
	func_block.RST := RST ;
	func_block.MIN_ONTIME := MIN_ONTIME;
	func_block.MIN_OFFTIME := MIN_OFFTIME;
	func_block.RUN_EVERY := RUN_EVERY ;
	func_block();
	PUMP  := func_block.PUMP;
	RUNTIME  := func_block.RUNTIME;
	CYCLES  := func_block.CYCLES;
END_PROGRAM

CONFIGURATION Config0
	VAR_GLOBAL
		PLC_TICKS_PER_SEC :	INT;
		PLC_SYS_TICK_CNT :	DINT;
	END_VAR
  	RESOURCE Res0 ON PLC
    	TASK task0(INTERVAL := T#20ms,PRIORITY := 0);
    	PROGRAM instance0 WITH task0 : program0;
  	END_RESOURCE
END_CONFIGURATION

(* ---- ACTUATOR_UD.ST ---- *)
FUNCTION_BLOCK T_PLC_MS_block
	VAR_OUTPUT
		T_PLC_MS :	UDINT;
	END_VAR

	VAR_EXTERNAL
		PLC_TICKS_PER_SEC :	INT;
		PLC_SYS_TICK_CNT :	DINT;
	END_VAR

	VAR
		debug :	BOOL;(*Debug-Mode ON / OFF*)
		N :	INT;(*Debug-Faktor*)
		Offset :	UDINT;(*Debug-Offset*)
		temp :	DWORD := DWORD#1;(*Debug-Offset*)
		mode :	BOOL;(*modus*)
		faktor :	UDINT;(*Systemtakt-Faktor*)
		init :	BOOL;
		v_plc_ticks_per_sec :	UDINT;
		base :	UDINT := UDINT#1000;
	END_VAR

	IF init = FALSE THEN
		v_plc_ticks_per_sec := INT_TO_UDINT(PLC_TICKS_PER_SEC);
		IF v_plc_ticks_per_sec = UDINT#1024 THEN
			faktor := UDINT#1;
			mode := FALSE;
		ELSIF v_plc_ticks_per_sec > UDINT#0 THEN
			IF v_plc_ticks_per_sec <= base THEN
				faktor := base / v_plc_ticks_per_sec;
				mode := FALSE;
			ELSE
				faktor := v_plc_ticks_per_sec / base;
				mode := TRUE;
			END_IF;
		ELSE
			faktor := UDINT#1;
		END_IF;
		init := TRUE;
	END_IF;

	IF mode THEN
		T_PLC_MS := DINT_TO_UDINT(PLC_SYS_TICK_CNT) / faktor;
	ELSE
		T_PLC_MS := DINT_TO_UDINT(PLC_SYS_TICK_CNT) * faktor;
	END_IF;

	IF debug THEN
		T_PLC_MS := (DWORD_TO_UDINT(SHL(UDINT_TO_DWORD(T_PLC_MS),N) OR SHL(temp,N)) - UDINT#1) + Offset;
	END_IF;
END_FUNCTION_BLOCK

FUNCTION_BLOCK ACTUATOR_UD_Block

	VAR_INPUT
		UD :	BOOL;
		_ON :	BOOL;
		MANUAL :	BOOL;
		UP :	BOOL;
		DN :	BOOL;
		OFF :	BOOL;
		YUP_IN :	BOOL;
		YDN_IN :	BOOL;
		_TON :	TIME;
		TOFF :	TIME;
		OUT_RETURN :	BOOL;
	END_VAR

	VAR_OUTPUT
		YUP :	BOOL;
		YDN :	BOOL;
		STATUS :	BYTE;
	END_VAR

	VAR
		tx :	TIME;
		last :	TIME;
		init :	BOOL;
		T_PLC_MS :	T_PLC_MS_Block;
	END_VAR

	T_PLC_MS();
	tx:= UDINT_TO_TIME(T_PLC_MS.T_PLC_MS);

	IF NOT init THEN
		last := tx;
		init := TRUE;
	ELSIF off THEN
		Yup := FALSE;
		Ydn := FALSE;
		last := tx;
		status := BYTE#101;

	ELSIF ((Yup OR Ydn) AND tx - last < _TON) THEN RETURN;
	ELSIF NOT yup AND NOT ydn AND tx - last < toff THEN	RETURN;

	ELSIF manual THEN
		status := BYTE#102;
		IF yup AND NOT up OR ydn AND NOT dn THEN
			ydn := FALSE;
			yup := FALSE;
			last := tx;
		ELSIF UP AND NOT DN AND NOT OFF THEN
			Ydn := FALSE;
			Yup := TRUE;
			last := tx;
			status := BYTE#103;
		ELSIF DN AND NOT UP AND NOT OFF THEN
			Yup := FALSE;
			Ydn := TRUE;
			last := tx;
			status := BYTE#104;
		ELSE
			IF YUP OR YDN THEN LAST := tx; END_IF;
			Yup := FALSE;
			Ydn := FALSE;
		END_IF;

	ELSE
		IF yup AND NOT ud OR ydn AND UD THEN
			yup := FALSE;
			ydn := FALSE;
			last := tx;
		ELSIF Ud AND _ON AND NOT OFF THEN
			Ydn := FALSE;
			Yup := TRUE;
			last := tx;
			status := BYTE#111;

		ELSIF NOT UD AND _ON AND NOT OFF THEN
			Yup := FALSE;
			Ydn := TRUE;
			last := tx;
			status := BYTE#112;
		ELSE
			IF Yup OR Ydn THEN last := tx; END_IF;
			Yup := FALSE;
			Ydn := FALSE;
			status := BYTE#110;
		END_IF;
	END_IF;

	IF Ydn AND Yup_in AND out_return THEN
		Ydn := FALSE;
		status := BYTE#1;
	END_IF;
	IF Yup AND Ydn_in AND out_return THEN
		Yup := FALSE;
		status := BYTE#2;
	END_IF;

END_FUNCTION_BLOCK

PROGRAM program0
	VAR
		UD :	BOOL;
		_ON :	BOOL;
		MANUAL :	BOOL;
		UP :	BOOL;
		DN :	BOOL;
		OFF :	BOOL;
		YUP_IN :	BOOL;
		YDN_IN :	BOOL;
		_TON :	TIME;
		TOFF :	TIME;
		OUT_RETURN :	BOOL;
		YUP :	BOOL;
		YDN :	BOOL;
		STATUS :	BYTE;
		func_block : ACTUATOR_UD_Block;
	END_VAR
	func_block.UD := UD;
	func_block._ON := _ON;
	func_block.MANUAL := MANUAL ;
	func_block.UP := UP;
	func_block.DN := DN;
	func_block.OFF := OFF ;
	func_block.YUP_IN := YUP_IN;
	func_block.YDN_IN := YDN_IN;
	func_block._TON := _TON ;
	func_block.TOFF := TOFF;
	func_block.OUT_RETURN := OUT_RETURN;
	func_block();
	YUP  := func_block.YUP;
	YDN  := func_block.YDN;
	STATUS  := func_block.STATUS;
END_PROGRAM

CONFIGURATION Config0
	VAR_GLOBAL
		PLC_TICKS_PER_SEC :	INT;
		PLC_SYS_TICK_CNT :	DINT;
	END_VAR
  	RESOURCE Res0 ON PLC
    	TASK task0(INTERVAL := T#20ms,PRIORITY := 0);
    	PROGRAM instance0 WITH task0 : program0;
  	END_RESOURCE
END_CONFIGURATION

(* ---- AIN1.ST ---- *)
FUNCTION_BLOCK AIN1

	VAR_INPUT
		IN :	DWORD;
		SIGN_BIT :	INT := 255;
		ERROR_BIT :	INT := 255;
		ERROR_CODE_EN :	BOOL := FALSE;
		ERROR_CODE :	DWORD;
		OVERFLOW_BIT :	INT := 255;
		OVERFLOW_CODE_EN :	BOOL;
		OVERFLOW_CODE :	DWORD;
		BIT_0 :	INT;
		BIT_N :	INT := 31;
		OUT_MIN :	REAL;
		OUT_MAX :	REAL := 10.0;
		CODE_MIN :	DWORD;
		CODE_MAX :	DWORD := DWORD#16#FFFFFFFF;
		ERROR_OUTPUT :	REAL;
		OVERFLOW_OUTPUT :	REAL := 10.0;
	END_VAR

	VAR_OUTPUT
		OUT :	REAL;
		SIGN :	BOOL;
		ERROR :	BOOL;
		OVERFLOW :	BOOL;
	END_VAR

	VAR
		tB :	DWORD;
	END_VAR

	error := ((SHR(in,error_bit) AND DWORD#16#0000_0001) = DWORD#1) OR (error_code_en AND error_code = in);
	IF error THEN
		out := error_output;
		RETURN;
	END_IF;

	tb := SHR(SHL(in, 31 - bit_N), 31 - bit_N + Bit_0);

	overflow := ((SHR(in,overflow_bit) AND DWORD#16#0000_0001) = DWORD#1) OR (overflow_code_en AND overflow_code = in) OR (tb < code_min OR tb > code_max);
	IF overflow THEN
		out := overflow_output;
		RETURN;
	END_IF;

	sign := (SHR(in,sign_bit) AND DWORD#16#0000_0001) = DWORD#1;

	out := (UDINT_TO_REAL(DWORD_TO_UDINT(tb) - DWORD_TO_UDINT(code_min)) * (out_max - out_min) / UDINT_TO_REAL(DWORD_TO_UDINT(code_max) - DWORD_TO_UDINT(code_min)) + out_min);
	IF sign THEN out := out * -1.0; END_IF;

	(* extract error bit *)
	error := ((SHR(in,error_bit) AND DWORD#16#0000_0001) = DWORD#1) OR (error_code_en AND error_code = in);
	IF error THEN
		out := error_output;
		RETURN;
	END_IF;

	(* strip off the data input *)
	tb := SHR(SHL(in, 31 - bit_N), 31 - bit_N + Bit_0);

	(* extract overflow bit *)
	overflow := ((SHR(in,overflow_bit) AND DWORD#16#0000_0001) = DWORD#1) OR (overflow_code_en AND overflow_code = in) OR (tb < code_min OR tb > code_max);
	IF overflow THEN
		out := overflow_output;
		RETURN;
	END_IF;

	(* extract sign bit *)
	sign := (SHR(in,sign_bit) AND DWORD#16#0000_0001) = DWORD#1;

	(* convert in to out *)
	out := (UDINT_TO_REAL(DWORD_TO_UDINT(tb) - DWORD_TO_UDINT(code_min)) * (out_max - out_min) / UDINT_TO_REAL(DWORD_TO_UDINT(code_max) - DWORD_TO_UDINT(code_min)) + out_min);
	IF sign THEN out := out * - 1.0; END_IF;

END_FUNCTION_BLOCK

PROGRAM program0
  VAR
	IN               :	DWORD;
	SIGN_BIT         :	INT ;
	ERROR_BIT        :	INT ;
	ERROR_CODE_EN    :	BOOL ;
	ERROR_CODE       :	DWORD;
	OVERFLOW_BIT     :	INT ;
	OVERFLOW_CODE_EN :	BOOL;
	OVERFLOW_CODE    :	DWORD;
	BIT_0            :	INT;
	BIT_N            :	INT;
	OUT_MIN          :	REAL;
	OUT_MAX          :	REAL ;
	CODE_MIN         :	DWORD;
	CODE_MAX         :	DWORD ;
	ERROR_OUTPUT     :	REAL;
	OVERFLOW_OUTPUT  :	REAL ;

	OUT      :	REAL;
	SIGN     :	BOOL;
	ERROR    :	BOOL;
	OVERFLOW :	BOOL;

	func_block : AIN1;
  END_VAR
	func_block.IN               :=IN              ;
	func_block.SIGN_BIT         :=SIGN_BIT        ;
	func_block.ERROR_BIT        :=ERROR_BIT       ;
	func_block.ERROR_CODE_EN    :=ERROR_CODE_EN   ;
	func_block.ERROR_CODE       :=ERROR_CODE      ;
	func_block.OVERFLOW_BIT     :=OVERFLOW_BIT    ;
	func_block.OVERFLOW_CODE_EN :=OVERFLOW_CODE_EN;
	func_block.OVERFLOW_CODE    :=OVERFLOW_CODE   ;
	func_block.BIT_0            :=BIT_0           ;
	func_block.BIT_N            :=BIT_N           ;
	func_block.OUT_MIN          :=OUT_MIN         ;
	func_block.OUT_MAX          :=OUT_MAX         ;
	func_block.CODE_MIN         :=CODE_MIN        ;
	func_block.CODE_MAX         :=CODE_MAX        ;
	func_block.ERROR_OUTPUT     :=ERROR_OUTPUT    ;
	func_block.OVERFLOW_OUTPUT  :=OVERFLOW_OUTPUT ;

	func_block();
	OUT     := func_block.OUT     ;
	SIGN    := func_block.SIGN    ;
	ERROR   := func_block.ERROR   ;
	OVERFLOW:= func_block.OVERFLOW;
END_PROGRAM

CONFIGURATION Config0
  RESOURCE Res0 ON PLC
    TASK task0(INTERVAL := T#20ms,PRIORITY := 0);
    PROGRAM instance0 WITH task0 : program0;
  END_RESOURCE
END_CONFIGURATION

(* ---- ALARM_2.ST ---- *)
FUNCTION_BLOCK ALARM_2
	VAR_INPUT
		X :	REAL;
		LO_1 :	REAL;
		HI_1 :	REAL;
		LO_2 :	REAL;
		HI_2 :	REAL;
		HYS :	REAL;
	END_VAR

	VAR_OUTPUT
		Q1_LO :	BOOL;
		Q1_HI :	BOOL;
		Q2_LO :	BOOL;
		Q2_HI :	BOOL;
	END_VAR

	VAR
		tmp :	REAL;
	END_VAR

	tmp := X - Hys * 0.5;
	IF tmp > LO_1 THEN Q1_LO := FALSE; END_IF;
	IF tmp > LO_2 THEN Q2_LO := FALSE; END_IF;
	IF tmp > HI_1 THEN Q1_HI := TRUE; END_IF;
	IF tmp > HI_2 THEN Q2_HI := TRUE; END_IF;
	tmp := tmp + hys;
	IF tmp < LO_1 THEN Q1_LO := TRUE; END_IF;
	IF tmp < LO_2 THEN Q2_LO := TRUE; END_IF;
	IF tmp < HI_1 THEN Q1_HI := FALSE; END_IF;
	IF tmp < HI_2 THEN Q2_HI := FALSE; END_IF;

END_FUNCTION_BLOCK

PROGRAM program0
	VAR
	    LocalVar0 : REAL;
		LocalVar1 : REAL;
		LocalVar2 : REAL;
		LocalVar3 : REAL;
		LocalVar4 : REAL;
		LocalVar5 : REAL;
		LocalOUT1  : BOOL;
		LocalOUT2  : BOOL;
		LocalOUT3  : BOOL;
		LocalOUT4  : BOOL;
		func_block : ALARM_2;
  	END_VAR
	func_block.X := LocalVar0;
	func_block.LO_1 := LocalVar1;
	func_block.HI_1 := LocalVar2;
	func_block.LO_2 := LocalVar3;
	func_block.HI_2 := LocalVar4;
	func_block.HYS := LocalVar5;
	func_block();
	LocalOUT1 := func_block.Q1_LO;
	LocalOUT2 := func_block.Q1_HI;
	LocalOUT3 := func_block.Q2_LO;
	LocalOUT4 := func_block.Q2_HI;
END_PROGRAM

CONFIGURATION Config0
  	RESOURCE Res0 ON PLC
    	TASK task0(INTERVAL := T#20ms,PRIORITY := 0);
    	PROGRAM instance0 WITH task0 : program0;
  	END_RESOURCE
END_CONFIGURATION

(* ---- ARRAY_AVG.ST ---- *)
TYPE
	oscat_pt_ARRAY: ARRAY [1..100] OF REAL;
END_TYPE

FUNCTION_BLOCK ARRAY_AVG_Block
	VAR_IN_OUT
		PT :	oscat_pt_ARRAY;
	END_VAR

	VAR_INPUT
		SIZE :	UINT;
	END_VAR

	VAR_OUTPUT
		ARRAY_AVG :	REAL;
	END_VAR

	VAR
		i :	INT;
		stop :	INT;
	END_VAR

	stop :=LIMIT_INT(1,UINT_TO_INT(size),1000);

	array_avg := 0.0;
	FOR i := 1 TO stop DO
		array_avg := array_avg + pt[i];
	END_FOR;
	array_avg := array_avg / INT_TO_REAL(stop);
END_FUNCTION_BLOCK

PROGRAM program0
  VAR
    LocalVar0 : oscat_pt_ARRAY;
    LocalVar1 : UINT;
	LocalOUT  : REAL;
	func_block : ARRAY_AVG_Block;
  END_VAR
	func_block.pt := LocalVar0;
	func_block.size := LocalVar1;
	func_block();
	LocalOUT := func_block.ARRAY_AVG;

END_PROGRAM

CONFIGURATION Config0
  RESOURCE Res0 ON PLC
    TASK task0(INTERVAL := T#20ms,PRIORITY := 0);
    PROGRAM instance0 WITH task0 : program0;
  END_RESOURCE
END_CONFIGURATION

(* ---- ARRAY_GAV.ST ---- *)
TYPE
	oscat_pt_ARRAY: ARRAY [1..100] OF REAL;
END_TYPE

FUNCTION SQRTN:REAL
	VAR_INPUT
		X :	REAL;
		N :	INT;
	END_VAR

	IF N > 0 THEN
		SQRTN := EXP(LN(x) / INT_TO_REAL(n));
	ELSE
		SQRTN := 0.0;
	END_IF;
END_FUNCTION

FUNCTION_BLOCK ARRAY_GAV_Block
	VAR_IN_OUT
		PT :	oscat_pt_ARRAY;
	END_VAR

	VAR_INPUT
		SIZE :	UINT;
	END_VAR

	VAR_OUTPUT
		ARRAY_GAV :	REAL;
	END_VAR

	VAR
		i :	INT;
		stop :	INT;
	END_VAR

	stop :=LIMIT_INT(1,UINT_TO_INT(size),1000);
	ARRAY_GAV := 1.0;
	FOR i := 1 TO stop DO
		IF pt[i] > 0.0 THEN
			ARRAY_GAV := ARRAY_GAV * pt[i];
		ELSE
			ARRAY_GAV := 0.0;
			RETURN;
		END_IF;
	END_FOR;
	ARRAY_GAV := SQRTN(ARRAY_GAV,stop);
END_FUNCTION_BLOCK

PROGRAM program0
  VAR
    LocalVar0 : oscat_pt_ARRAY;
    LocalVar1 : UINT;
	LocalOUT  : REAL;
	func_block : ARRAY_GAV_Block;
  END_VAR
	func_block.pt := LocalVar0;
	func_block.size := LocalVar1;
	func_block();
	LocalOUT := func_block.ARRAY_GAV;

END_PROGRAM

CONFIGURATION Config0
  RESOURCE Res0 ON PLC
    TASK task0(INTERVAL := T#20ms,PRIORITY := 0);
    PROGRAM instance0 WITH task0 : program0;
  END_RESOURCE
END_CONFIGURATION

(* ---- ARRAY_HAV.ST ---- *)
TYPE
	oscat_pt_ARRAY: ARRAY [1..100] OF REAL;
END_TYPE

FUNCTION_BLOCK ARRAY_HAV_Block
	VAR_IN_OUT
		PT :	oscat_pt_ARRAY;
	END_VAR

	VAR_INPUT
		SIZE :	UINT;
	END_VAR

	VAR_OUTPUT
		ARRAY_HAV :	REAL;
	END_VAR

	VAR
		i :	INT;
		stop :	INT;
	END_VAR

	stop :=LIMIT_INT(1,UINT_TO_INT(size),1000);
	ARRAY_HAV := 0.0;
	FOR i := 1 TO stop DO
		IF pt[i] <> 0.0 THEN
			ARRAY_HAV := ARRAY_HAV + 1.0/pt[i];
		ELSE
			ARRAY_HAV := 0.0;
			RETURN;
		END_IF;
	END_FOR;
	ARRAY_HAV := INT_TO_REAL(stop) / ARRAY_HAV;
END_FUNCTION_BLOCK

PROGRAM program0
  VAR
    LocalVar0 : oscat_pt_ARRAY;
    LocalVar1 : UINT;
	LocalOUT  : REAL;
	func_block : ARRAY_HAV_Block;
  END_VAR
	func_block.pt := LocalVar0;
	func_block.size := LocalVar1;
	func_block();
	LocalOUT := func_block.ARRAY_HAV;

END_PROGRAM

CONFIGURATION Config0
  RESOURCE Res0 ON PLC
    TASK task0(INTERVAL := T#20ms,PRIORITY := 0);
    PROGRAM instance0 WITH task0 : program0;
  END_RESOURCE
END_CONFIGURATION

(* ---- ARRAY_MAX.ST ---- *)
TYPE
	oscat_pt_ARRAY: ARRAY [1..100] OF REAL;
END_TYPE

FUNCTION_BLOCK ARRAY_MAX_Block
	VAR_IN_OUT
		PT :	oscat_pt_ARRAY;
	END_VAR

	VAR_INPUT
		SIZE :	UINT;
	END_VAR

	VAR_OUTPUT
		ARRAY_MAX :	REAL;
	END_VAR

	VAR
		i :	INT;
		stop :	INT;
	END_VAR

	stop :=LIMIT_INT(1,UINT_TO_INT(size),1000);

	FOR i := 1 TO stop DO
		IF pt[i] > array_max THEN array_max := pt[i]; END_IF;
	END_FOR;

END_FUNCTION_BLOCK

PROGRAM program0
  VAR
    LocalVar0 : oscat_pt_ARRAY;
    LocalVar1 : UINT;
	LocalOUT  : REAL;
	func_block : ARRAY_MAX_Block;
  END_VAR
	func_block.pt := LocalVar0;
	func_block.size := LocalVar1;
	func_block();
	LocalOUT := func_block.ARRAY_MAX;

END_PROGRAM

CONFIGURATION Config0
  RESOURCE Res0 ON PLC
    TASK task0(INTERVAL := T#20ms,PRIORITY := 0);
    PROGRAM instance0 WITH task0 : program0;
  END_RESOURCE
END_CONFIGURATION

(* ---- ARRAY_MEDIAN.ST ---- *)
TYPE
	oscat_pt_ARRAY: ARRAY [1..100] OF REAL;
	oscat_stack_array: ARRAY [1..32]   OF INT;
END_TYPE

FUNCTION _INT_TO_UDINT:UDINT
	VAR_INPUT
		IN :	INT;
	END_VAR

	_INT_TO_UDINT := DINT_TO_UDINT(INT_TO_DINT(IN));
END_FUNCTION

FUNCTION BIT_OF_DWORD:BOOL
	VAR_INPUT
		IN :	DWORD;
		N :	INT;
	END_VAR
	BIT_OF_DWORD := (SHR(in,n) AND DWORD#1) > DWORD#0;
END_FUNCTION

FUNCTION EVEN:BOOL
	VAR_INPUT
		IN :	DINT;
	END_VAR
	even := NOT BIT_OF_DWORD(DINT_TO_DWORD(in),0);
END_FUNCTION

FUNCTION_BLOCK _ARRAY_SORT_Block
	VAR_IN_OUT
		PT :	oscat_pt_ARRAY;
	END_VAR

	VAR_INPUT
		SIZE :	UINT;
	END_VAR

	VAR_OUTPUT
		_ARRAY_SORT :BOOL;
	END_VAR

	VAR
		stack_count :	INT;
		stack :	oscat_stack_array;
		links :	INT;
		rechts :	INT;
		pivot :	REAL;
		i :	INT;
		j :	INT;
		ende_innen :	BOOL;
		ende_aussen :	BOOL;
		tmp :	REAL;
		x :	INT;
	END_VAR

	links := 1;
	rechts := DWORD_TO_INT(SHR(UINT_TO_DWORD(size),2));
	stack_count := 1;

	WHILE NOT ende_aussen DO
		IF links < rechts THEN
			x := DWORD_TO_INT(SHR(UDINT_TO_DWORD(_INT_TO_UDINT(rechts)+ _INT_TO_UDINT(links)),1));
			pivot := PT[x];
			i := links - 1;
			j := rechts + 1;

			ende_innen := FALSE;
			REPEAT
				REPEAT	i := i+1;	UNTIL (PT[i] >= pivot) OR NOT (i < rechts)	END_REPEAT;
				REPEAT	j := j-1;	UNTIL (PT[j] <= pivot) OR NOT (j > links)	END_REPEAT;
				IF i >= j THEN
					ende_innen := TRUE;
				ELSE
					tmp := PT[j];
					PT[j] := PT[i];
					PT[i] := tmp;
				END_IF;

			UNTIL ende_innen END_REPEAT;

			stack[stack_count] := rechts;
			IF Stack_count < 32 THEN
				stack_count := stack_count +1;
			ELSE
				ende_aussen := TRUE;
				_ARRAY_SORT := FALSE;
			END_IF;
			rechts := MAX(links, i-1);

		ELSE
			IF stack_count = 1 THEN
				ende_aussen := TRUE;
			ELSE
				links := rechts+1;
				stack_count := stack_count - 1;
				rechts:= stack[stack_count];
			END_IF;
		END_IF;
	END_WHILE;

	_ARRAY_SORT := TRUE;
END_FUNCTION_BLOCK

FUNCTION_BLOCK _ARRAY_MEDIAN_Block

	VAR_IN_OUT
		PT :	oscat_pt_ARRAY;
	END_VAR

	VAR_INPUT
		SIZE :	UINT;
	END_VAR

	VAR_OUTPUT
		_ARRAY_MEDIAN :	REAL;
	END_VAR

	VAR
		i :	INT;
		i2 :	INT;
		stop :	INT;
		_array_sort :	_ARRAY_SORT_Block;
	END_VAR

	(* Array sortieren *)
	_array_sort.pt   := pt;
	_array_sort.size := size;
	_array_sort();
	pt := _array_sort.pt;

	stop :=LIMIT_INT(1,UINT_TO_INT(size),1000);
	IF even(INT_TO_DINT(stop)) THEN
	    i := WORD_TO_INT(SHR(INT_TO_WORD(stop),1));
	    i2 := i+1;
		_array_median := (pt[i] + pt[i2]) * 0.5;
	ELSE
	    i := WORD_TO_INT(SHR(INT_TO_WORD(stop),1))+1;
		_array_median := pt[i];
	END_IF;

END_FUNCTION_BLOCK

PROGRAM program0
  VAR
    LocalVar0 : oscat_pt_ARRAY;
    LocalVar1 : UINT;
	LocalOUT  : REAL;
	func_block : _ARRAY_MEDIAN_Block;
  END_VAR
	func_block.pt := LocalVar0;
	func_block.size := LocalVar1;
	func_block();
	LocalOUT := func_block._ARRAY_MEDIAN;
	LocalVar0 := func_block.pt;

END_PROGRAM

CONFIGURATION Config0
  RESOURCE Res0 ON PLC
    TASK task0(INTERVAL := T#20ms,PRIORITY := 0);
    PROGRAM instance0 WITH task0 : program0;
  END_RESOURCE
END_CONFIGURATION

(* ---- ARRAY_MIN.ST ---- *)
TYPE
	oscat_pt_ARRAY: ARRAY [1..100] OF REAL;
END_TYPE

FUNCTION_BLOCK ARRAY_MIN_Block
	VAR_IN_OUT
		PT :	oscat_pt_ARRAY;
	END_VAR

	VAR_INPUT
		SIZE :	UINT;
	END_VAR

	VAR_OUTPUT
		ARRAY_MIN :	REAL;
	END_VAR

	VAR
		i :	INT;
		stop :	INT;
	END_VAR

	stop :=LIMIT_INT(1,UINT_TO_INT(size),1000);

	array_min := pt[1];
	FOR i := 2 TO stop DO
		IF pt[i] < array_min THEN array_min := pt[i]; END_IF;
	END_FOR;

END_FUNCTION_BLOCK
PROGRAM program0
  VAR
    LocalVar0 : oscat_pt_ARRAY;
    LocalVar1 : UINT;
	LocalOUT  : REAL;
	func_block : ARRAY_MIN_Block;
  END_VAR
	func_block.pt := LocalVar0;
	func_block.size := LocalVar1;
	func_block();
	LocalOUT := func_block.ARRAY_MIN;

END_PROGRAM

CONFIGURATION Config0
  RESOURCE Res0 ON PLC
    TASK task0(INTERVAL := T#20ms,PRIORITY := 0);
    PROGRAM instance0 WITH task0 : program0;
  END_RESOURCE
END_CONFIGURATION

(* ---- ARRAY_SDV.ST ---- *)
TYPE
	oscat_pt_ARRAY: ARRAY [1..100] OF REAL;
END_TYPE

FUNCTION_BLOCK ARRAY_VAR_Block
	VAR_IN_OUT
		PT :	oscat_pt_ARRAY;
	END_VAR

	VAR_INPUT
		SIZE :	UINT;
	END_VAR

	VAR_OUTPUT
		ARRAY_VAR :	REAL;
	END_VAR

	VAR
		i :	INT;
		stop :	INT;
		avg :	REAL;
	END_VAR

	stop :=LIMIT_INT(1,UINT_TO_INT(size),1000);
	avg := pt[1];
	FOR i := 2 TO stop DO
		avg := avg + pt[i];
	END_FOR;
	avg := avg / INT_TO_REAL(stop);

	array_var := EXPT(pt[1] - avg, 2.0);
	FOR i := 2 TO stop DO
		array_var := array_var + EXPT(pt[i] - avg, 2.0);
	END_FOR;
	array_var := array_var / INT_TO_REAL(stop-1);

END_FUNCTION_BLOCK

FUNCTION_BLOCK ARRAY_SDV_Block
	VAR_IN_OUT
		PT :	oscat_pt_ARRAY;
	END_VAR

	VAR_INPUT
		SIZE :	UINT;
	END_VAR

	VAR_OUTPUT
		ARRAY_SDV :	REAL;
	END_VAR

	VAR
		FB_array_var :	array_var_block;
	END_VAR

	FB_array_var.pt   := pt;
	FB_array_var.size := size;
	FB_array_var();
	pt := FB_array_var.pt;

	array_sdv := SQRT(FB_array_var.array_var);
END_FUNCTION_BLOCK

PROGRAM program0
  VAR
    LocalVar0 : oscat_pt_ARRAY;
    LocalVar1 : UINT;
	LocalOUT  : REAL;
	func_block : ARRAY_SDV_Block;
  END_VAR
	func_block.pt := LocalVar0;
	func_block.size := LocalVar1;
	func_block();
	LocalOUT := func_block.ARRAY_SDV;

END_PROGRAM

CONFIGURATION Config0
  RESOURCE Res0 ON PLC
    TASK task0(INTERVAL := T#20ms,PRIORITY := 0);
    PROGRAM instance0 WITH task0 : program0;
  END_RESOURCE
END_CONFIGURATION

(* ---- ARRAY_SPR.ST ---- *)
TYPE
	oscat_pt_ARRAY: ARRAY [1..100] OF REAL;
END_TYPE

FUNCTION_BLOCK ARRAY_SPR_Block
	VAR_IN_OUT
		PT :	oscat_pt_ARRAY;
	END_VAR

	VAR_INPUT
		SIZE :	UINT;
	END_VAR

	VAR_OUTPUT
		ARRAY_SPR :	REAL;
	END_VAR

	VAR
		i :	INT;
		stop :	INT;
		array_max :	REAL;
		array_min :	REAL;
	END_VAR

	stop :=LIMIT_INT(1,UINT_TO_INT(size),1000);

	array_min := pt[1];
	array_max := pt[1];
	FOR i := 2 TO stop DO
		IF pt[i] > array_max THEN array_max := pt[i];
		ELSIF pt[i] < array_min THEN array_min := pt[i];
		END_IF;
	END_FOR;
	array_spr := array_max - array_min;
END_FUNCTION_BLOCK

PROGRAM program0
  VAR
    LocalVar0 : oscat_pt_ARRAY;
    LocalVar1 : UINT;
	LocalOUT  : REAL;
	func_block : ARRAY_SPR_Block;
  END_VAR
	func_block.pt := LocalVar0;
	func_block.size := LocalVar1;
	func_block();
	LocalOUT := func_block.ARRAY_SPR;

END_PROGRAM

CONFIGURATION Config0
  RESOURCE Res0 ON PLC
    TASK task0(INTERVAL := T#20ms,PRIORITY := 0);
    PROGRAM instance0 WITH task0 : program0;
  END_RESOURCE
END_CONFIGURATION

(* ---- ARRAY_SUM.ST ---- *)
TYPE
	oscat_pt_ARRAY: ARRAY [1..100] OF REAL;
END_TYPE

FUNCTION_BLOCK ARRAY_SUM_Block
	VAR_IN_OUT
		PT :	oscat_pt_ARRAY;
	END_VAR

	VAR_INPUT
		SIZE :	UINT;
	END_VAR

	VAR_OUTPUT
		ARRAY_SUM :	REAL;
	END_VAR

	VAR
		i :	INT;
		stop :	INT;
	END_VAR

	stop :=LIMIT_INT(1,UINT_TO_INT(size),1000);

	array_sum := pt[1];
	FOR i := 2 TO stop DO
		array_sum := array_sum + pt[i];
	END_FOR;
END_FUNCTION_BLOCK

PROGRAM program0
  VAR
    LocalVar0 : oscat_pt_ARRAY;
    LocalVar1 : UINT;
	LocalOUT  : REAL;
	func_block : ARRAY_SUM_Block;
  END_VAR
	func_block.pt := LocalVar0;
	func_block.size := LocalVar1;
	func_block();
	LocalOUT := func_block.ARRAY_SUM;

END_PROGRAM

CONFIGURATION Config0
  RESOURCE Res0 ON PLC
    TASK task0(INTERVAL := T#20ms,PRIORITY := 0);
    PROGRAM instance0 WITH task0 : program0;
  END_RESOURCE
END_CONFIGURATION

(* ---- ARRAY_TREND.ST ---- *)
TYPE
	oscat_pt_ARRAY: ARRAY [1..100] OF REAL;
END_TYPE

FUNCTION BIT_OF_DWORD:BOOL
	VAR_INPUT
		IN :	DWORD;
		N :	INT;
	END_VAR
	BIT_OF_DWORD := (SHR(in,n) AND DWORD#1) > DWORD#0;
END_FUNCTION

FUNCTION EVEN:BOOL
	VAR_INPUT
		IN :	DINT;
	END_VAR
	even := NOT BIT_OF_DWORD(DINT_TO_DWORD(in),0);
END_FUNCTION

FUNCTION_BLOCK ARRAY_TREND_Block
	VAR_IN_OUT
		PT :	oscat_pt_ARRAY;
	END_VAR

	VAR_INPUT
		SIZE :	UINT;
	END_VAR

	VAR_OUTPUT
		ARRAY_TREND :	REAL;
	END_VAR

	VAR
		d :	INT;
		i :	INT;
		stop :	INT;
		stop2 :	INT;
		x :	REAL;
	END_VAR

	x := 0.0;
	stop :=LIMIT_INT(1,UINT_TO_INT(size),1000);
	stop2 := WORD_TO_INT(SHR(INT_TO_WORD(stop),1));
	IF even(INT_TO_DINT(stop)) THEN d:=0; ELSE d:=1;END_IF;

	FOR i := 1 TO stop2+d DO
		x := x - pt[i];
	END_FOR;
	FOR i := stop2+1 TO stop DO
		x := x + pt[i];
	END_FOR;
	array_trend := x / INT_TO_REAL(stop2+d);

END_FUNCTION_BLOCK

PROGRAM program0
  VAR
    LocalVar0 : oscat_pt_ARRAY;
    LocalVar1 : UINT;
	LocalOUT  : REAL;
	func_block : ARRAY_TREND_Block;
  END_VAR
	func_block.pt := LocalVar0;
	func_block.size := LocalVar1;
	func_block();
	LocalOUT := func_block.ARRAY_TREND;

END_PROGRAM

CONFIGURATION Config0
  RESOURCE Res0 ON PLC
    TASK task0(INTERVAL := T#20ms,PRIORITY := 0);
    PROGRAM instance0 WITH task0 : program0;
  END_RESOURCE
END_CONFIGURATION

(* ---- ARRAY_VAR.ST ---- *)
TYPE
	oscat_pt_ARRAY: ARRAY [1..100] OF REAL;
END_TYPE

FUNCTION_BLOCK ARRAY_VAR_Block
	VAR_IN_OUT
		PT :	oscat_pt_ARRAY;
	END_VAR

	VAR_INPUT
		SIZE :	UINT;
	END_VAR

	VAR_OUTPUT
		ARRAY_VAR :	REAL;
	END_VAR

	VAR
		i :	INT;
		stop :	INT;
		avg :	REAL;
	END_VAR

	stop :=LIMIT_INT(1,UINT_TO_INT(size),1000);
	avg := pt[1];
	FOR i := 2 TO stop DO
		avg := avg + pt[i];
	END_FOR;
	avg := avg / INT_TO_REAL(stop);

	array_var := EXPT(pt[1] - avg, 2.0);
	FOR i := 2 TO stop DO
		array_var := array_var + EXPT(pt[i] - avg, 2.0);
	END_FOR;
	array_var := array_var / INT_TO_REAL(stop-1);

END_FUNCTION_BLOCK

PROGRAM program0
  VAR
    LocalVar0 : oscat_pt_ARRAY;
    LocalVar1 : UINT;
	LocalOUT  : REAL;
	func_block : ARRAY_VAR_Block;
  END_VAR
	func_block.pt := LocalVar0;
	func_block.size := LocalVar1;
	func_block();
	LocalOUT := func_block.ARRAY_VAR;

END_PROGRAM

CONFIGURATION Config0
  RESOURCE Res0 ON PLC
    TASK task0(INTERVAL := T#20ms,PRIORITY := 0);
    PROGRAM instance0 WITH task0 : program0;
  END_RESOURCE
END_CONFIGURATION

(* ---- ASTRO.ST ---- *)
FUNCTION_BLOCK ASTRO
	VAR_INPUT
		M :	REAL;
		AE :	REAL;
		PC :	REAL;
		LJ :	REAL;
	END_VAR

	VAR_OUTPUT
		YM :	REAL;
		YAE :	REAL;
		YPC :	REAL;
		YLJ :	REAL;
	END_VAR

	YAE :=	AE
			+ m * 6.6845871535E-012
			+ PC * 206265.0
			+ LJ * 63240.0;
	Ym := YAE * 149.597870E9;
	YPC := YAE * 4.8481322570E-006;
	YLJ := YAE * 1.5812776724E-005;
END_FUNCTION_BLOCK

PROGRAM program0
  VAR
    LocalVar0 : REAL;
    LocalVar1 : REAL;
	LocalVar2 : REAL;
	LocalVar3 : REAL;
	LocalOUT1 : REAL;
	LocalOUT2 : REAL;
	LocalOUT3 : REAL;
	LocalOUT4 : REAL;
	func_block : ASTRO;
  END_VAR
	func_block.M  := LocalVar0;
	func_block.AE := LocalVar1;
	func_block.PC := LocalVar2;
	func_block.LJ := LocalVar3;
	func_block();
	LocalOUT1 := func_block.YM ;
	LocalOUT2 := func_block.YAE;
	LocalOUT3 := func_block.YPC;
	LocalOUT4 := func_block.YLJ;

END_PROGRAM

CONFIGURATION Config0
  RESOURCE Res0 ON PLC
    TASK task0(INTERVAL := T#20ms,PRIORITY := 0);
    PROGRAM instance0 WITH task0 : program0;
  END_RESOURCE
END_CONFIGURATION

(* ---- AUTORUN.ST ---- *)
FUNCTION UDINT_TO_TIME2:TIME

	VAR_INPUT
		IN :	UDINT;
	END_VAR

	UDINT_TO_TIME2 := DINT_TO_TIME(UDINT_TO_DINT(IN));

END_FUNCTION

FUNCTION_BLOCK T_PLC_MS_block
	VAR_OUTPUT
		T_PLC_MS :	UDINT;
	END_VAR

	VAR_EXTERNAL
		PLC_TICKS_PER_SEC :	INT;
		PLC_SYS_TICK_CNT :	DINT;
	END_VAR

	VAR
		debug :	BOOL;(*Debug-Mode ON / OFF*)
		N :	INT;(*Debug-Faktor*)
		Offset :	UDINT;(*Debug-Offset*)
		temp :	DWORD := DWORD#1;(*Debug-Offset*)
		mode :	BOOL;(*modus*)
		faktor :	UDINT;(*Systemtakt-Faktor*)
		init :	BOOL;
		v_plc_ticks_per_sec :	UDINT;
		base :	UDINT := UDINT#1000;
	END_VAR

	IF init = FALSE THEN
		v_plc_ticks_per_sec := INT_TO_UDINT(PLC_TICKS_PER_SEC);
		IF v_plc_ticks_per_sec = UDINT#1024 THEN
			faktor := UDINT#1;
			mode := FALSE;
		ELSIF v_plc_ticks_per_sec > UDINT#0 THEN
			IF v_plc_ticks_per_sec <= base THEN
				faktor := base / v_plc_ticks_per_sec;
				mode := FALSE;
			ELSE
				faktor := v_plc_ticks_per_sec / base;
				mode := TRUE;
			END_IF;
		ELSE
			faktor := UDINT#1;
		END_IF;
		init := TRUE;
	END_IF;

	IF mode THEN
		T_PLC_MS := DINT_TO_UDINT(PLC_SYS_TICK_CNT) / faktor;
	ELSE
		T_PLC_MS := DINT_TO_UDINT(PLC_SYS_TICK_CNT) * faktor;
	END_IF;

	IF debug THEN
		T_PLC_MS := (DWORD_TO_UDINT(SHL(UDINT_TO_DWORD(T_PLC_MS),N) OR SHL(temp,N)) - UDINT#1) + Offset;
	END_IF;

END_FUNCTION_BLOCK

FUNCTION TIME_TO_UDINT2:UDINT
	VAR_INPUT
		X :	TIME;
	END_VAR

	TIME_TO_UDINT2 := DINT_TO_UDINT(TIME_TO_DINT(X));
END_FUNCTION

FUNCTION FRMP_B:BYTE
	VAR_INPUT
		START :	BYTE;
		DIR :	BOOL;
		TD :	TIME;
		TR :	TIME;
	END_VAR

	IF TD < TR THEN
		FRMP_B := MIN(UDINT_TO_BYTE(DWORD_TO_UDINT(SHL(TIME_TO_DWORD(TD), 8)) / TIME_TO_UDINT2(TR)), SEL(DIR, START, USINT_TO_BYTE(USINT#255 - BYTE_TO_USINT(START))));
		IF DIR THEN
			FRMP_B := USINT_TO_BYTE(BYTE_TO_USINT(START) + BYTE_TO_USINT(FRMP_B));
		ELSE
			FRMP_B := USINT_TO_BYTE(BYTE_TO_USINT(START) - BYTE_TO_USINT(FRMP_B));
		END_IF;
	ELSE
		FRMP_B := SEL(DIR, BYTE#0, BYTE#255);
	END_IF;
END_FUNCTION

FUNCTION_BLOCK _RMP_B
	VAR_INPUT
		DIR :	BOOL;
		E :	BOOL := TRUE;
		TR :	TIME;
	END_VAR

	VAR_IN_OUT
		RMP :	BYTE;
	END_VAR

	VAR
		T_PLC_MS :	T_PLC_MS_block;
		tx :	TIME;
		tl :	TIME;
		tn :	TIME;
		init :	BOOL;
		last_dir :	BOOL;
		start :	BYTE;
	END_VAR

	T_PLC_MS();
	tx := UDINT_TO_TIME(T_PLC_MS.T_PLC_MS);

	IF E AND init AND (dir = last_dir) AND (RMP <> SEL(DIR, BYTE#0, BYTE#255)) AND TR = tn THEN
		RMP := FRMP_B(start, DIR, tx - tl, TR);
	ELSE
		init := TRUE;
		tl := tx;
		tn := tr;
		start := RMP;
	END_IF;
	last_dir := dir;
END_FUNCTION_BLOCK

FUNCTION_BLOCK AUTORUN_Block

	VAR_INPUT
		IN :	BOOL;
		TEST :	BOOL;
		ARE :	BOOL := TRUE;
		TRUN :	TIME;
		TOFF :	TIME;
	END_VAR

	VAR_OUTPUT
		OUT :	BOOL;
		ARO :	BOOL;
	END_VAR

	VAR_IN_OUT
		ARX :	BOOL;
	END_VAR

	VAR
		timer :	_RMP_B;
		val :	BYTE;
	END_VAR

	IF TOFF > T#0s THEN
		timer(DIR:= OUT, TR := SEL(OUT, TOFF, TRUN), RMP := val);
		val := timer.RMP;
	ELSE
		val := BYTE#255;
	END_IF;

	IF (NOT ARX AND ARE AND val = BYTE#0) OR TEST THEN
		val := BYTE#0;
		ARO := TRUE;
		ARX := TRUE;
	ELSIF val = BYTE#255 AND ARO THEN
		ARO := FALSE;
		ARX := FALSE;
	END_IF;

	out := IN OR ARO;

END_FUNCTION_BLOCK

PROGRAM program0
	VAR
		IN :	BOOL;
		TEST :	BOOL;
		ARE :	BOOL := TRUE;
		TRUN :	TIME;
		TOFF :	TIME;
		OUT :	BOOL;
		ARO :	BOOL;
		func_block : AUTORUN_Block;
	END_VAR
	func_block.IN := IN;
	func_block.TEST := TEST;
	func_block.ARE := ARE ;
	func_block.TRUN := TRUN;
	func_block.TOFF := TOFF;
	func_block();
	OUT  := func_block.OUT;
	ARO  := func_block.ARO;
END_PROGRAM

CONFIGURATION Config0
	VAR_GLOBAL
		PLC_TICKS_PER_SEC :	INT;
		PLC_SYS_TICK_CNT :	DINT;
	END_VAR
  	RESOURCE Res0 ON PLC
    	TASK task0(INTERVAL := T#20ms,PRIORITY := 0);
    	PROGRAM instance0 WITH task0 : program0;
  	END_RESOURCE
END_CONFIGURATION

(* ---- B_TRIG.ST ---- *)
FUNCTION_BLOCK B_TRIG
	VAR_INPUT
		CLK :	BOOL;
	END_VAR

	VAR_OUTPUT
		Q :	BOOL := FALSE;
	END_VAR

	VAR
		edge :	BOOL := FALSE;
	END_VAR

	Q := clk XOR edge;
	edge := CLK;
END_FUNCTION_BLOCK

PROGRAM program0
  VAR
    LocalVar0 : BOOL;
	LocalOUT  : BOOL;
	func_block : B_TRIG;
  END_VAR
	func_block.CLK := LocalVar0;
	func_block();
	LocalOUT := func_block.Q;

END_PROGRAM

CONFIGURATION Config0
  RESOURCE Res0 ON PLC
    TASK task0(INTERVAL := T#20ms,PRIORITY := 0);
    PROGRAM instance0 WITH task0 : program0;
  END_RESOURCE
END_CONFIGURATION
